    CONST robtarget point_414_contact:=[[206,145,134.5],[0,0,1,0],[0, 0, 0, 0],[9E+09,9E+09,9E+09,9E+09,9E+09,9E+09]];
    CONST robtarget point_415_contact:=[[206,137,134.5],[0,0,1,0],[0, 0, 0, 0],[9E+09,9E+09,9E+09,9E+09,9E+09,9E+09]];
    CONST robtarget point_415_clearance:=[[206,137,149.5],[0,0,1,0],[0, 0, 0, 0],[9E+09,9E+09,9E+09,9E+09,9E+09,9E+09]];
    CONST robtarget point_416_clearance:=[[237,138,149.5],[0,0,1,0],[0, 0, 0, 0],[9E+09,9E+09,9E+09,9E+09,9E+09,9E+09]];
    CONST robtarget point_416_contact:=[[237,138,134.5],[0,0,1,0],[0, 0, 0, 0],[9E+09,9E+09,9E+09,9E+09,9E+09,9E+09]];
    CONST robtarget point_417_contact:=[[240,137,134.5],[0,0,1,0],[0, 0, 0, 0],[9E+09,9E+09,9E+09,9E+09,9E+09,9E+09]];
    CONST robtarget point_417_clearance:=[[240,137,149.5],[0,0,1,0],[0, 0, 0, 0],[9E+09,9E+09,9E+09,9E+09,9E+09,9E+09]];
    CONST robtarget point_418_clearance:=[[348,137,149.5],[0,0,1,0],[0, 0, 0, 0],[9E+09,9E+09,9E+09,9E+09,9E+09,9E+09]];
    CONST robtarget point_418_contact:=[[348,137,134.5],[0,0,1,0],[0, 0, 0, 0],[9E+09,9E+09,9E+09,9E+09,9E+09,9E+09]];
    CONST robtarget point_419_contact:=[[363,145,134.5],[0,0,1,0],[0, 0, 0, 0],[9E+09,9E+09,9E+09,9E+09,9E+09,9E+09]];
    CONST robtarget point_419_clearance:=[[363,145,149.5],[0,0,1,0],[0, 0, 0, 0],[9E+09,9E+09,9E+09,9E+09,9E+09,9E+09]];
    CONST robtarget point_420_clearance:=[[399,156,149.5],[0,0,1,0],[0, 0, 0, 0],[9E+09,9E+09,9E+09,9E+09,9E+09,9E+09]];
    CONST robtarget point_420_contact:=[[399,156,134.5],[0,0,1,0],[0, 0, 0, 0],[9E+09,9E+09,9E+09,9E+09,9E+09,9E+09]];
    CONST robtarget point_421_contact:=[[402,137,134.5],[0,0,1,0],[0, 0, 0, 0],[9E+09,9E+09,9E+09,9E+09,9E+09,9E+09]];
    CONST robtarget point_421_clearance:=[[402,137,149.5],[0,0,1,0],[0, 0, 0, 0],[9E+09,9E+09,9E+09,9E+09,9E+09,9E+09]];
    CONST robtarget point_422_clearance:=[[144,140,149.5],[0,0,1,0],[0, 0, 0, 0],[9E+09,9E+09,9E+09,9E+09,9E+09,9E+09]];
    CONST robtarget point_422_contact:=[[144,140,134.5],[0,0,1,0],[0, 0, 0, 0],[9E+09,9E+09,9E+09,9E+09,9E+09,9E+09]];
    CONST robtarget point_423_contact:=[[159,145,134.5],[0,0,1,0],[0, 0, 0, 0],[9E+09,9E+09,9E+09,9E+09,9E+09,9E+09]];
    CONST robtarget point_423_clearance:=[[159,145,149.5],[0,0,1,0],[0, 0, 0, 0],[9E+09,9E+09,9E+09,9E+09,9E+09,9E+09]];
    CONST robtarget point_424_clearance:=[[249,145,149.5],[0,0,1,0],[0, 0, 0, 0],[9E+09,9E+09,9E+09,9E+09,9E+09,9E+09]];
    CONST robtarget point_424_contact:=[[249,145,134.5],[0,0,1,0],[0, 0, 0, 0],[9E+09,9E+09,9E+09,9E+09,9E+09,9E+09]];
    CONST robtarget point_425_contact:=[[256,139,134.5],[0,0,1,0],[0, 0, 0, 0],[9E+09,9E+09,9E+09,9E+09,9E+09,9E+09]];
    CONST robtarget point_425_clearance:=[[256,139,149.5],[0,0,1,0],[0, 0, 0, 0],[9E+09,9E+09,9E+09,9E+09,9E+09,9E+09]];
    CONST robtarget point_426_clearance:=[[316,140,149.5],[0,0,1,0],[0, 0, 0, 0],[9E+09,9E+09,9E+09,9E+09,9E+09,9E+09]];
    CONST robtarget point_426_contact:=[[316,140,134.5],[0,0,1,0],[0, 0, 0, 0],[9E+09,9E+09,9E+09,9E+09,9E+09,9E+09]];
    CONST robtarget point_427_contact:=[[312,141,134.5],[0,0,1,0],[0, 0, 0, 0],[9E+09,9E+09,9E+09,9E+09,9E+09,9E+09]];
    CONST robtarget point_427_clearance:=[[312,141,149.5],[0,0,1,0],[0, 0, 0, 0],[9E+09,9E+09,9E+09,9E+09,9E+09,9E+09]];
    CONST robtarget point_428_clearance:=[[313,144,149.5],[0,0,1,0],[0, 0, 0, 0],[9E+09,9E+09,9E+09,9E+09,9E+09,9E+09]];
    CONST robtarget point_428_contact:=[[313,144,134.5],[0,0,1,0],[0, 0, 0, 0],[9E+09,9E+09,9E+09,9E+09,9E+09,9E+09]];
    CONST robtarget point_429_contact:=[[322,138,134.5],[0,0,1,0],[0, 0, 0, 0],[9E+09,9E+09,9E+09,9E+09,9E+09,9E+09]];
    CONST robtarget point_429_clearance:=[[322,138,149.5],[0,0,1,0],[0, 0, 0, 0],[9E+09,9E+09,9E+09,9E+09,9E+09,9E+09]];
    CONST robtarget point_430_clearance:=[[368,140,149.5],[0,0,1,0],[0, 0, 0, 0],[9E+09,9E+09,9E+09,9E+09,9E+09,9E+09]];
    CONST robtarget point_430_contact:=[[368,140,134.5],[0,0,1,0],[0, 0, 0, 0],[9E+09,9E+09,9E+09,9E+09,9E+09,9E+09]];
    CONST robtarget point_431_contact:=[[371,139,134.5],[0,0,1,0],[0, 0, 0, 0],[9E+09,9E+09,9E+09,9E+09,9E+09,9E+09]];
    CONST robtarget point_431_clearance:=[[371,139,149.5],[0,0,1,0],[0, 0, 0, 0],[9E+09,9E+09,9E+09,9E+09,9E+09,9E+09]];
    CONST robtarget point_432_clearance:=[[306,146,149.5],[0,0,1,0],[0, 0, 0, 0],[9E+09,9E+09,9E+09,9E+09,9E+09,9E+09]];
    CONST robtarget point_432_contact:=[[306,146,134.5],[0,0,1,0],[0, 0, 0, 0],[9E+09,9E+09,9E+09,9E+09,9E+09,9E+09]];
    CONST robtarget point_433_contact:=[[299,140,134.5],[0,0,1,0],[0, 0, 0, 0],[9E+09,9E+09,9E+09,9E+09,9E+09,9E+09]];
    CONST robtarget point_433_clearance:=[[299,140,149.5],[0,0,1,0],[0, 0, 0, 0],[9E+09,9E+09,9E+09,9E+09,9E+09,9E+09]];
    CONST robtarget point_434_clearance:=[[411,141,149.5],[0,0,1,0],[0, 0, 0, 0],[9E+09,9E+09,9E+09,9E+09,9E+09,9E+09]];
    CONST robtarget point_434_contact:=[[411,141,134.5],[0,0,1,0],[0, 0, 0, 0],[9E+09,9E+09,9E+09,9E+09,9E+09,9E+09]];
    CONST robtarget point_435_contact:=[[409,155,134.5],[0,0,1,0],[0, 0, 0, 0],[9E+09,9E+09,9E+09,9E+09,9E+09,9E+09]];
    CONST robtarget point_435_clearance:=[[409,155,149.5],[0,0,1,0],[0, 0, 0, 0],[9E+09,9E+09,9E+09,9E+09,9E+09,9E+09]];
    CONST robtarget point_436_clearance:=[[160,143,149.5],[0,0,1,0],[0, 0, 0, 0],[9E+09,9E+09,9E+09,9E+09,9E+09,9E+09]];
    CONST robtarget point_436_contact:=[[160,143,134.5],[0,0,1,0],[0, 0, 0, 0],[9E+09,9E+09,9E+09,9E+09,9E+09,9E+09]];
    CONST robtarget point_437_contact:=[[160,162,134.5],[0,0,1,0],[0, 0, 0, 0],[9E+09,9E+09,9E+09,9E+09,9E+09,9E+09]];
    CONST robtarget point_437_clearance:=[[160,162,149.5],[0,0,1,0],[0, 0, 0, 0],[9E+09,9E+09,9E+09,9E+09,9E+09,9E+09]];
    CONST robtarget point_438_clearance:=[[316,147,149.5],[0,0,1,0],[0, 0, 0, 0],[9E+09,9E+09,9E+09,9E+09,9E+09,9E+09]];
    CONST robtarget point_438_contact:=[[316,147,134.5],[0,0,1,0],[0, 0, 0, 0],[9E+09,9E+09,9E+09,9E+09,9E+09,9E+09]];
    CONST robtarget point_439_contact:=[[306,146,134.5],[0,0,1,0],[0, 0, 0, 0],[9E+09,9E+09,9E+09,9E+09,9E+09,9E+09]];
    CONST robtarget point_439_clearance:=[[306,146,149.5],[0,0,1,0],[0, 0, 0, 0],[9E+09,9E+09,9E+09,9E+09,9E+09,9E+09]];
    CONST robtarget point_440_clearance:=[[435,170,149.5],[0,0,1,0],[0, 0, 0, 0],[9E+09,9E+09,9E+09,9E+09,9E+09,9E+09]];
    CONST robtarget point_440_contact:=[[435,170,134.5],[0,0,1,0],[0, 0, 0, 0],[9E+09,9E+09,9E+09,9E+09,9E+09,9E+09]];
    CONST robtarget point_441_contact:=[[433,143,134.5],[0,0,1,0],[0, 0, 0, 0],[9E+09,9E+09,9E+09,9E+09,9E+09,9E+09]];
    CONST robtarget point_441_clearance:=[[433,143,149.5],[0,0,1,0],[0, 0, 0, 0],[9E+09,9E+09,9E+09,9E+09,9E+09,9E+09]];
    CONST robtarget point_442_clearance:=[[326,146,149.5],[0,0,1,0],[0, 0, 0, 0],[9E+09,9E+09,9E+09,9E+09,9E+09,9E+09]];
    CONST robtarget point_442_contact:=[[326,146,134.5],[0,0,1,0],[0, 0, 0, 0],[9E+09,9E+09,9E+09,9E+09,9E+09,9E+09]];
    CONST robtarget point_443_contact:=[[317,146,134.5],[0,0,1,0],[0, 0, 0, 0],[9E+09,9E+09,9E+09,9E+09,9E+09,9E+09]];
    CONST robtarget point_443_clearance:=[[317,146,149.5],[0,0,1,0],[0, 0, 0, 0],[9E+09,9E+09,9E+09,9E+09,9E+09,9E+09]];
    CONST robtarget point_444_clearance:=[[378,183,149.5],[0,0,1,0],[0, 0, 0, 0],[9E+09,9E+09,9E+09,9E+09,9E+09,9E+09]];
    CONST robtarget point_444_contact:=[[378,183,134.5],[0,0,1,0],[0, 0, 0, 0],[9E+09,9E+09,9E+09,9E+09,9E+09,9E+09]];
    CONST robtarget point_445_contact:=[[391,144,134.5],[0,0,1,0],[0, 0, 0, 0],[9E+09,9E+09,9E+09,9E+09,9E+09,9E+09]];
    CONST robtarget point_445_clearance:=[[391,144,149.5],[0,0,1,0],[0, 0, 0, 0],[9E+09,9E+09,9E+09,9E+09,9E+09,9E+09]];
    CONST robtarget point_446_clearance:=[[166,147,149.5],[0,0,1,0],[0, 0, 0, 0],[9E+09,9E+09,9E+09,9E+09,9E+09,9E+09]];
    CONST robtarget point_446_contact:=[[166,147,134.5],[0,0,1,0],[0, 0, 0, 0],[9E+09,9E+09,9E+09,9E+09,9E+09,9E+09]];
    CONST robtarget point_447_contact:=[[176,150,134.5],[0,0,1,0],[0, 0, 0, 0],[9E+09,9E+09,9E+09,9E+09,9E+09,9E+09]];
    CONST robtarget point_447_clearance:=[[176,150,149.5],[0,0,1,0],[0, 0, 0, 0],[9E+09,9E+09,9E+09,9E+09,9E+09,9E+09]];
    CONST robtarget point_448_clearance:=[[198,172,149.5],[0,0,1,0],[0, 0, 0, 0],[9E+09,9E+09,9E+09,9E+09,9E+09,9E+09]];
    CONST robtarget point_448_contact:=[[198,172,134.5],[0,0,1,0],[0, 0, 0, 0],[9E+09,9E+09,9E+09,9E+09,9E+09,9E+09]];
    CONST robtarget point_449_contact:=[[198,146,134.5],[0,0,1,0],[0, 0, 0, 0],[9E+09,9E+09,9E+09,9E+09,9E+09,9E+09]];
    CONST robtarget point_449_clearance:=[[198,146,149.5],[0,0,1,0],[0, 0, 0, 0],[9E+09,9E+09,9E+09,9E+09,9E+09,9E+09]];
    CONST robtarget point_450_clearance:=[[213,226,149.5],[0,0,1,0],[0, 0, 0, 0],[9E+09,9E+09,9E+09,9E+09,9E+09,9E+09]];
    CONST robtarget point_450_contact:=[[213,226,134.5],[0,0,1,0],[0, 0, 0, 0],[9E+09,9E+09,9E+09,9E+09,9E+09,9E+09]];
    CONST robtarget point_451_contact:=[[206,146,134.5],[0,0,1,0],[0, 0, 0, 0],[9E+09,9E+09,9E+09,9E+09,9E+09,9E+09]];
    CONST robtarget point_451_clearance:=[[206,146,149.5],[0,0,1,0],[0, 0, 0, 0],[9E+09,9E+09,9E+09,9E+09,9E+09,9E+09]];
    CONST robtarget point_452_clearance:=[[165,163,149.5],[0,0,1,0],[0, 0, 0, 0],[9E+09,9E+09,9E+09,9E+09,9E+09,9E+09]];
    CONST robtarget point_452_contact:=[[165,163,134.5],[0,0,1,0],[0, 0, 0, 0],[9E+09,9E+09,9E+09,9E+09,9E+09,9E+09]];
    CONST robtarget point_453_contact:=[[165,150,134.5],[0,0,1,0],[0, 0, 0, 0],[9E+09,9E+09,9E+09,9E+09,9E+09,9E+09]];
    CONST robtarget point_453_clearance:=[[165,150,149.5],[0,0,1,0],[0, 0, 0, 0],[9E+09,9E+09,9E+09,9E+09,9E+09,9E+09]];
    CONST robtarget point_454_clearance:=[[188,150,149.5],[0,0,1,0],[0, 0, 0, 0],[9E+09,9E+09,9E+09,9E+09,9E+09,9E+09]];
    CONST robtarget point_454_contact:=[[188,150,134.5],[0,0,1,0],[0, 0, 0, 0],[9E+09,9E+09,9E+09,9E+09,9E+09,9E+09]];
    CONST robtarget point_455_contact:=[[188,170,134.5],[0,0,1,0],[0, 0, 0, 0],[9E+09,9E+09,9E+09,9E+09,9E+09,9E+09]];
    CONST robtarget point_455_clearance:=[[188,170,149.5],[0,0,1,0],[0, 0, 0, 0],[9E+09,9E+09,9E+09,9E+09,9E+09,9E+09]];
    CONST robtarget point_456_clearance:=[[230,150,149.5],[0,0,1,0],[0, 0, 0, 0],[9E+09,9E+09,9E+09,9E+09,9E+09,9E+09]];
    CONST robtarget point_456_contact:=[[230,150,134.5],[0,0,1,0],[0, 0, 0, 0],[9E+09,9E+09,9E+09,9E+09,9E+09,9E+09]];
    CONST robtarget point_457_contact:=[[237,168,134.5],[0,0,1,0],[0, 0, 0, 0],[9E+09,9E+09,9E+09,9E+09,9E+09,9E+09]];
    CONST robtarget point_457_clearance:=[[237,168,149.5],[0,0,1,0],[0, 0, 0, 0],[9E+09,9E+09,9E+09,9E+09,9E+09,9E+09]];
    CONST robtarget point_458_clearance:=[[266,154,149.5],[0,0,1,0],[0, 0, 0, 0],[9E+09,9E+09,9E+09,9E+09,9E+09,9E+09]];
    CONST robtarget point_458_contact:=[[266,154,134.5],[0,0,1,0],[0, 0, 0, 0],[9E+09,9E+09,9E+09,9E+09,9E+09,9E+09]];
    CONST robtarget point_459_contact:=[[343,158,134.5],[0,0,1,0],[0, 0, 0, 0],[9E+09,9E+09,9E+09,9E+09,9E+09,9E+09]];
    CONST robtarget point_459_clearance:=[[343,158,149.5],[0,0,1,0],[0, 0, 0, 0],[9E+09,9E+09,9E+09,9E+09,9E+09,9E+09]];
    CONST robtarget point_460_clearance:=[[357,162,149.5],[0,0,1,0],[0, 0, 0, 0],[9E+09,9E+09,9E+09,9E+09,9E+09,9E+09]];
    CONST robtarget point_460_contact:=[[357,162,134.5],[0,0,1,0],[0, 0, 0, 0],[9E+09,9E+09,9E+09,9E+09,9E+09,9E+09]];
    CONST robtarget point_461_contact:=[[344,149,134.5],[0,0,1,0],[0, 0, 0, 0],[9E+09,9E+09,9E+09,9E+09,9E+09,9E+09]];
    CONST robtarget point_461_clearance:=[[344,149,149.5],[0,0,1,0],[0, 0, 0, 0],[9E+09,9E+09,9E+09,9E+09,9E+09,9E+09]];
    CONST robtarget point_462_clearance:=[[179,151,149.5],[0,0,1,0],[0, 0, 0, 0],[9E+09,9E+09,9E+09,9E+09,9E+09,9E+09]];
    CONST robtarget point_462_contact:=[[179,151,134.5],[0,0,1,0],[0, 0, 0, 0],[9E+09,9E+09,9E+09,9E+09,9E+09,9E+09]];
    CONST robtarget point_463_contact:=[[179,167,134.5],[0,0,1,0],[0, 0, 0, 0],[9E+09,9E+09,9E+09,9E+09,9E+09,9E+09]];
    CONST robtarget point_463_clearance:=[[179,167,149.5],[0,0,1,0],[0, 0, 0, 0],[9E+09,9E+09,9E+09,9E+09,9E+09,9E+09]];
    CONST robtarget point_464_clearance:=[[413,187,149.5],[0,0,1,0],[0, 0, 0, 0],[9E+09,9E+09,9E+09,9E+09,9E+09,9E+09]];
    CONST robtarget point_464_contact:=[[413,187,134.5],[0,0,1,0],[0, 0, 0, 0],[9E+09,9E+09,9E+09,9E+09,9E+09,9E+09]];
    CONST robtarget point_465_contact:=[[415,151,134.5],[0,0,1,0],[0, 0, 0, 0],[9E+09,9E+09,9E+09,9E+09,9E+09,9E+09]];
    CONST robtarget point_465_clearance:=[[415,151,149.5],[0,0,1,0],[0, 0, 0, 0],[9E+09,9E+09,9E+09,9E+09,9E+09,9E+09]];
    CONST robtarget point_466_clearance:=[[257,154,149.5],[0,0,1,0],[0, 0, 0, 0],[9E+09,9E+09,9E+09,9E+09,9E+09,9E+09]];
    CONST robtarget point_466_contact:=[[257,154,134.5],[0,0,1,0],[0, 0, 0, 0],[9E+09,9E+09,9E+09,9E+09,9E+09,9E+09]];
    CONST robtarget point_467_contact:=[[241,160,134.5],[0,0,1,0],[0, 0, 0, 0],[9E+09,9E+09,9E+09,9E+09,9E+09,9E+09]];
    CONST robtarget point_467_clearance:=[[241,160,149.5],[0,0,1,0],[0, 0, 0, 0],[9E+09,9E+09,9E+09,9E+09,9E+09,9E+09]];
    CONST robtarget point_468_clearance:=[[260,158,149.5],[0,0,1,0],[0, 0, 0, 0],[9E+09,9E+09,9E+09,9E+09,9E+09,9E+09]];
    CONST robtarget point_468_contact:=[[260,158,134.5],[0,0,1,0],[0, 0, 0, 0],[9E+09,9E+09,9E+09,9E+09,9E+09,9E+09]];
    CONST robtarget point_469_contact:=[[265,153,134.5],[0,0,1,0],[0, 0, 0, 0],[9E+09,9E+09,9E+09,9E+09,9E+09,9E+09]];
    CONST robtarget point_469_clearance:=[[265,153,149.5],[0,0,1,0],[0, 0, 0, 0],[9E+09,9E+09,9E+09,9E+09,9E+09,9E+09]];
    CONST robtarget point_470_clearance:=[[410,154,149.5],[0,0,1,0],[0, 0, 0, 0],[9E+09,9E+09,9E+09,9E+09,9E+09,9E+09]];
    CONST robtarget point_470_contact:=[[410,154,134.5],[0,0,1,0],[0, 0, 0, 0],[9E+09,9E+09,9E+09,9E+09,9E+09,9E+09]];
    CONST robtarget point_471_contact:=[[398,192,134.5],[0,0,1,0],[0, 0, 0, 0],[9E+09,9E+09,9E+09,9E+09,9E+09,9E+09]];
    CONST robtarget point_471_clearance:=[[398,192,149.5],[0,0,1,0],[0, 0, 0, 0],[9E+09,9E+09,9E+09,9E+09,9E+09,9E+09]];
    CONST robtarget point_472_clearance:=[[161,164,149.5],[0,0,1,0],[0, 0, 0, 0],[9E+09,9E+09,9E+09,9E+09,9E+09,9E+09]];
    CONST robtarget point_472_contact:=[[161,164,134.5],[0,0,1,0],[0, 0, 0, 0],[9E+09,9E+09,9E+09,9E+09,9E+09,9E+09]];
    CONST robtarget point_473_contact:=[[145,159,134.5],[0,0,1,0],[0, 0, 0, 0],[9E+09,9E+09,9E+09,9E+09,9E+09,9E+09]];
    CONST robtarget point_473_clearance:=[[145,159,149.5],[0,0,1,0],[0, 0, 0, 0],[9E+09,9E+09,9E+09,9E+09,9E+09,9E+09]];
    CONST robtarget point_474_clearance:=[[191,182,149.5],[0,0,1,0],[0, 0, 0, 0],[9E+09,9E+09,9E+09,9E+09,9E+09,9E+09]];
    CONST robtarget point_474_contact:=[[191,182,134.5],[0,0,1,0],[0, 0, 0, 0],[9E+09,9E+09,9E+09,9E+09,9E+09,9E+09]];
    CONST robtarget point_475_contact:=[[192,157,134.5],[0,0,1,0],[0, 0, 0, 0],[9E+09,9E+09,9E+09,9E+09,9E+09,9E+09]];
    CONST robtarget point_475_clearance:=[[192,157,149.5],[0,0,1,0],[0, 0, 0, 0],[9E+09,9E+09,9E+09,9E+09,9E+09,9E+09]];
    CONST robtarget point_476_clearance:=[[218,178,149.5],[0,0,1,0],[0, 0, 0, 0],[9E+09,9E+09,9E+09,9E+09,9E+09,9E+09]];
    CONST robtarget point_476_contact:=[[218,178,134.5],[0,0,1,0],[0, 0, 0, 0],[9E+09,9E+09,9E+09,9E+09,9E+09,9E+09]];
    CONST robtarget point_477_contact:=[[219,157,134.5],[0,0,1,0],[0, 0, 0, 0],[9E+09,9E+09,9E+09,9E+09,9E+09,9E+09]];
    CONST robtarget point_477_clearance:=[[219,157,149.5],[0,0,1,0],[0, 0, 0, 0],[9E+09,9E+09,9E+09,9E+09,9E+09,9E+09]];
    CONST robtarget point_478_clearance:=[[315,163,149.5],[0,0,1,0],[0, 0, 0, 0],[9E+09,9E+09,9E+09,9E+09,9E+09,9E+09]];
    CONST robtarget point_478_contact:=[[315,163,134.5],[0,0,1,0],[0, 0, 0, 0],[9E+09,9E+09,9E+09,9E+09,9E+09,9E+09]];
    CONST robtarget point_479_contact:=[[257,160,134.5],[0,0,1,0],[0, 0, 0, 0],[9E+09,9E+09,9E+09,9E+09,9E+09,9E+09]];
    CONST robtarget point_479_clearance:=[[257,160,149.5],[0,0,1,0],[0, 0, 0, 0],[9E+09,9E+09,9E+09,9E+09,9E+09,9E+09]];
    CONST robtarget point_480_clearance:=[[395,187,149.5],[0,0,1,0],[0, 0, 0, 0],[9E+09,9E+09,9E+09,9E+09,9E+09,9E+09]];
    CONST robtarget point_480_contact:=[[395,187,134.5],[0,0,1,0],[0, 0, 0, 0],[9E+09,9E+09,9E+09,9E+09,9E+09,9E+09]];
    CONST robtarget point_481_contact:=[[401,160,134.5],[0,0,1,0],[0, 0, 0, 0],[9E+09,9E+09,9E+09,9E+09,9E+09,9E+09]];
    CONST robtarget point_481_clearance:=[[401,160,149.5],[0,0,1,0],[0, 0, 0, 0],[9E+09,9E+09,9E+09,9E+09,9E+09,9E+09]];
    CONST robtarget point_482_clearance:=[[285,172,149.5],[0,0,1,0],[0, 0, 0, 0],[9E+09,9E+09,9E+09,9E+09,9E+09,9E+09]];
    CONST robtarget point_482_contact:=[[285,172,134.5],[0,0,1,0],[0, 0, 0, 0],[9E+09,9E+09,9E+09,9E+09,9E+09,9E+09]];
    CONST robtarget point_483_contact:=[[271,161,134.5],[0,0,1,0],[0, 0, 0, 0],[9E+09,9E+09,9E+09,9E+09,9E+09,9E+09]];
    CONST robtarget point_483_clearance:=[[271,161,149.5],[0,0,1,0],[0, 0, 0, 0],[9E+09,9E+09,9E+09,9E+09,9E+09,9E+09]];
    CONST robtarget point_484_clearance:=[[356,164,149.5],[0,0,1,0],[0, 0, 0, 0],[9E+09,9E+09,9E+09,9E+09,9E+09,9E+09]];
    CONST robtarget point_484_contact:=[[356,164,134.5],[0,0,1,0],[0, 0, 0, 0],[9E+09,9E+09,9E+09,9E+09,9E+09,9E+09]];
    CONST robtarget point_485_contact:=[[363,162,134.5],[0,0,1,0],[0, 0, 0, 0],[9E+09,9E+09,9E+09,9E+09,9E+09,9E+09]];
    CONST robtarget point_485_clearance:=[[363,162,149.5],[0,0,1,0],[0, 0, 0, 0],[9E+09,9E+09,9E+09,9E+09,9E+09,9E+09]];
    CONST robtarget point_486_clearance:=[[347,164,149.5],[0,0,1,0],[0, 0, 0, 0],[9E+09,9E+09,9E+09,9E+09,9E+09,9E+09]];
    CONST robtarget point_486_contact:=[[347,164,134.5],[0,0,1,0],[0, 0, 0, 0],[9E+09,9E+09,9E+09,9E+09,9E+09,9E+09]];
    CONST robtarget point_487_contact:=[[316,163,134.5],[0,0,1,0],[0, 0, 0, 0],[9E+09,9E+09,9E+09,9E+09,9E+09,9E+09]];
    CONST robtarget point_487_clearance:=[[316,163,149.5],[0,0,1,0],[0, 0, 0, 0],[9E+09,9E+09,9E+09,9E+09,9E+09,9E+09]];
    CONST robtarget point_488_clearance:=[[176,169,149.5],[0,0,1,0],[0, 0, 0, 0],[9E+09,9E+09,9E+09,9E+09,9E+09,9E+09]];
    CONST robtarget point_488_contact:=[[176,169,134.5],[0,0,1,0],[0, 0, 0, 0],[9E+09,9E+09,9E+09,9E+09,9E+09,9E+09]];
    CONST robtarget point_489_contact:=[[171,164,134.5],[0,0,1,0],[0, 0, 0, 0],[9E+09,9E+09,9E+09,9E+09,9E+09,9E+09]];
    CONST robtarget point_489_clearance:=[[171,164,149.5],[0,0,1,0],[0, 0, 0, 0],[9E+09,9E+09,9E+09,9E+09,9E+09,9E+09]];
    CONST robtarget point_490_clearance:=[[203,164,149.5],[0,0,1,0],[0, 0, 0, 0],[9E+09,9E+09,9E+09,9E+09,9E+09,9E+09]];
    CONST robtarget point_490_contact:=[[203,164,134.5],[0,0,1,0],[0, 0, 0, 0],[9E+09,9E+09,9E+09,9E+09,9E+09,9E+09]];
    CONST robtarget point_491_contact:=[[206,185,134.5],[0,0,1,0],[0, 0, 0, 0],[9E+09,9E+09,9E+09,9E+09,9E+09,9E+09]];
    CONST robtarget point_491_clearance:=[[206,185,149.5],[0,0,1,0],[0, 0, 0, 0],[9E+09,9E+09,9E+09,9E+09,9E+09,9E+09]];
    CONST robtarget point_492_clearance:=[[331,167,149.5],[0,0,1,0],[0, 0, 0, 0],[9E+09,9E+09,9E+09,9E+09,9E+09,9E+09]];
    CONST robtarget point_492_contact:=[[331,167,134.5],[0,0,1,0],[0, 0, 0, 0],[9E+09,9E+09,9E+09,9E+09,9E+09,9E+09]];
    CONST robtarget point_493_contact:=[[340,168,134.5],[0,0,1,0],[0, 0, 0, 0],[9E+09,9E+09,9E+09,9E+09,9E+09,9E+09]];
    CONST robtarget point_493_clearance:=[[340,168,149.5],[0,0,1,0],[0, 0, 0, 0],[9E+09,9E+09,9E+09,9E+09,9E+09,9E+09]];
    CONST robtarget point_494_clearance:=[[396,165,149.5],[0,0,1,0],[0, 0, 0, 0],[9E+09,9E+09,9E+09,9E+09,9E+09,9E+09]];
    CONST robtarget point_494_contact:=[[396,165,134.5],[0,0,1,0],[0, 0, 0, 0],[9E+09,9E+09,9E+09,9E+09,9E+09,9E+09]];
    CONST robtarget point_495_contact:=[[393,183,134.5],[0,0,1,0],[0, 0, 0, 0],[9E+09,9E+09,9E+09,9E+09,9E+09,9E+09]];
    CONST robtarget point_495_clearance:=[[393,183,149.5],[0,0,1,0],[0, 0, 0, 0],[9E+09,9E+09,9E+09,9E+09,9E+09,9E+09]];
    CONST robtarget point_496_clearance:=[[286,166,149.5],[0,0,1,0],[0, 0, 0, 0],[9E+09,9E+09,9E+09,9E+09,9E+09,9E+09]];
    CONST robtarget point_496_contact:=[[286,166,134.5],[0,0,1,0],[0, 0, 0, 0],[9E+09,9E+09,9E+09,9E+09,9E+09,9E+09]];
    CONST robtarget point_497_contact:=[[306,170,134.5],[0,0,1,0],[0, 0, 0, 0],[9E+09,9E+09,9E+09,9E+09,9E+09,9E+09]];
    CONST robtarget point_497_clearance:=[[306,170,149.5],[0,0,1,0],[0, 0, 0, 0],[9E+09,9E+09,9E+09,9E+09,9E+09,9E+09]];
    CONST robtarget point_498_clearance:=[[364,171,149.5],[0,0,1,0],[0, 0, 0, 0],[9E+09,9E+09,9E+09,9E+09,9E+09,9E+09]];
    CONST robtarget point_498_contact:=[[364,171,134.5],[0,0,1,0],[0, 0, 0, 0],[9E+09,9E+09,9E+09,9E+09,9E+09,9E+09]];
    CONST robtarget point_499_contact:=[[367,166,134.5],[0,0,1,0],[0, 0, 0, 0],[9E+09,9E+09,9E+09,9E+09,9E+09,9E+09]];
    CONST robtarget point_499_clearance:=[[367,166,149.5],[0,0,1,0],[0, 0, 0, 0],[9E+09,9E+09,9E+09,9E+09,9E+09,9E+09]];
    CONST robtarget point_500_clearance:=[[425,166,149.5],[0,0,1,0],[0, 0, 0, 0],[9E+09,9E+09,9E+09,9E+09,9E+09,9E+09]];
    CONST robtarget point_500_contact:=[[425,166,134.5],[0,0,1,0],[0, 0, 0, 0],[9E+09,9E+09,9E+09,9E+09,9E+09,9E+09]];
    CONST robtarget point_501_contact:=[[421,199,134.5],[0,0,1,0],[0, 0, 0, 0],[9E+09,9E+09,9E+09,9E+09,9E+09,9E+09]];
    CONST robtarget point_501_clearance:=[[421,199,149.5],[0,0,1,0],[0, 0, 0, 0],[9E+09,9E+09,9E+09,9E+09,9E+09,9E+09]];
    CONST robtarget point_502_clearance:=[[425,196,149.5],[0,0,1,0],[0, 0, 0, 0],[9E+09,9E+09,9E+09,9E+09,9E+09,9E+09]];
    CONST robtarget point_502_contact:=[[425,196,134.5],[0,0,1,0],[0, 0, 0, 0],[9E+09,9E+09,9E+09,9E+09,9E+09,9E+09]];
    CONST robtarget point_503_contact:=[[428,166,134.5],[0,0,1,0],[0, 0, 0, 0],[9E+09,9E+09,9E+09,9E+09,9E+09,9E+09]];
    CONST robtarget point_503_clearance:=[[428,166,149.5],[0,0,1,0],[0, 0, 0, 0],[9E+09,9E+09,9E+09,9E+09,9E+09,9E+09]];
    CONST robtarget point_504_clearance:=[[307,169,149.5],[0,0,1,0],[0, 0, 0, 0],[9E+09,9E+09,9E+09,9E+09,9E+09,9E+09]];
    CONST robtarget point_504_contact:=[[307,169,134.5],[0,0,1,0],[0, 0, 0, 0],[9E+09,9E+09,9E+09,9E+09,9E+09,9E+09]];
    CONST robtarget point_505_contact:=[[323,168,134.5],[0,0,1,0],[0, 0, 0, 0],[9E+09,9E+09,9E+09,9E+09,9E+09,9E+09]];
    CONST robtarget point_505_clearance:=[[323,168,149.5],[0,0,1,0],[0, 0, 0, 0],[9E+09,9E+09,9E+09,9E+09,9E+09,9E+09]];
    CONST robtarget point_506_clearance:=[[330,168,149.5],[0,0,1,0],[0, 0, 0, 0],[9E+09,9E+09,9E+09,9E+09,9E+09,9E+09]];
    CONST robtarget point_506_contact:=[[330,168,134.5],[0,0,1,0],[0, 0, 0, 0],[9E+09,9E+09,9E+09,9E+09,9E+09,9E+09]];
    CONST robtarget point_507_contact:=[[319,174,134.5],[0,0,1,0],[0, 0, 0, 0],[9E+09,9E+09,9E+09,9E+09,9E+09,9E+09]];
    CONST robtarget point_507_clearance:=[[319,174,149.5],[0,0,1,0],[0, 0, 0, 0],[9E+09,9E+09,9E+09,9E+09,9E+09,9E+09]];
    CONST robtarget point_508_clearance:=[[138,170,149.5],[0,0,1,0],[0, 0, 0, 0],[9E+09,9E+09,9E+09,9E+09,9E+09,9E+09]];
    CONST robtarget point_508_contact:=[[138,170,134.5],[0,0,1,0],[0, 0, 0, 0],[9E+09,9E+09,9E+09,9E+09,9E+09,9E+09]];
    CONST robtarget point_509_contact:=[[159,174,134.5],[0,0,1,0],[0, 0, 0, 0],[9E+09,9E+09,9E+09,9E+09,9E+09,9E+09]];
    CONST robtarget point_509_clearance:=[[159,174,149.5],[0,0,1,0],[0, 0, 0, 0],[9E+09,9E+09,9E+09,9E+09,9E+09,9E+09]];
    CONST robtarget point_510_clearance:=[[237,168,149.5],[0,0,1,0],[0, 0, 0, 0],[9E+09,9E+09,9E+09,9E+09,9E+09,9E+09]];
    CONST robtarget point_510_contact:=[[237,168,134.5],[0,0,1,0],[0, 0, 0, 0],[9E+09,9E+09,9E+09,9E+09,9E+09,9E+09]];
    CONST robtarget point_511_contact:=[[238,176,134.5],[0,0,1,0],[0, 0, 0, 0],[9E+09,9E+09,9E+09,9E+09,9E+09,9E+09]];
    CONST robtarget point_511_clearance:=[[238,176,149.5],[0,0,1,0],[0, 0, 0, 0],[9E+09,9E+09,9E+09,9E+09,9E+09,9E+09]];
    CONST robtarget point_512_clearance:=[[357,169,149.5],[0,0,1,0],[0, 0, 0, 0],[9E+09,9E+09,9E+09,9E+09,9E+09,9E+09]];
    CONST robtarget point_512_contact:=[[357,169,134.5],[0,0,1,0],[0, 0, 0, 0],[9E+09,9E+09,9E+09,9E+09,9E+09,9E+09]];
    CONST robtarget point_513_contact:=[[360,172,134.5],[0,0,1,0],[0, 0, 0, 0],[9E+09,9E+09,9E+09,9E+09,9E+09,9E+09]];
    CONST robtarget point_513_clearance:=[[360,172,149.5],[0,0,1,0],[0, 0, 0, 0],[9E+09,9E+09,9E+09,9E+09,9E+09,9E+09]];
    CONST robtarget point_514_clearance:=[[412,168,149.5],[0,0,1,0],[0, 0, 0, 0],[9E+09,9E+09,9E+09,9E+09,9E+09,9E+09]];
    CONST robtarget point_514_contact:=[[412,168,134.5],[0,0,1,0],[0, 0, 0, 0],[9E+09,9E+09,9E+09,9E+09,9E+09,9E+09]];
    CONST robtarget point_515_contact:=[[407,197,134.5],[0,0,1,0],[0, 0, 0, 0],[9E+09,9E+09,9E+09,9E+09,9E+09,9E+09]];
    CONST robtarget point_515_clearance:=[[407,197,149.5],[0,0,1,0],[0, 0, 0, 0],[9E+09,9E+09,9E+09,9E+09,9E+09,9E+09]];
    CONST robtarget point_516_clearance:=[[188,170,149.5],[0,0,1,0],[0, 0, 0, 0],[9E+09,9E+09,9E+09,9E+09,9E+09,9E+09]];
    CONST robtarget point_516_contact:=[[188,170,134.5],[0,0,1,0],[0, 0, 0, 0],[9E+09,9E+09,9E+09,9E+09,9E+09,9E+09]];
    CONST robtarget point_517_contact:=[[186,175,134.5],[0,0,1,0],[0, 0, 0, 0],[9E+09,9E+09,9E+09,9E+09,9E+09,9E+09]];
    CONST robtarget point_517_clearance:=[[186,175,149.5],[0,0,1,0],[0, 0, 0, 0],[9E+09,9E+09,9E+09,9E+09,9E+09,9E+09]];
    CONST robtarget point_518_clearance:=[[200,173,149.5],[0,0,1,0],[0, 0, 0, 0],[9E+09,9E+09,9E+09,9E+09,9E+09,9E+09]];
    CONST robtarget point_518_contact:=[[200,173,134.5],[0,0,1,0],[0, 0, 0, 0],[9E+09,9E+09,9E+09,9E+09,9E+09,9E+09]];
    CONST robtarget point_519_contact:=[[201,186,134.5],[0,0,1,0],[0, 0, 0, 0],[9E+09,9E+09,9E+09,9E+09,9E+09,9E+09]];
    CONST robtarget point_519_clearance:=[[201,186,149.5],[0,0,1,0],[0, 0, 0, 0],[9E+09,9E+09,9E+09,9E+09,9E+09,9E+09]];
    CONST robtarget point_520_clearance:=[[160,175,149.5],[0,0,1,0],[0, 0, 0, 0],[9E+09,9E+09,9E+09,9E+09,9E+09,9E+09]];
    CONST robtarget point_520_contact:=[[160,175,134.5],[0,0,1,0],[0, 0, 0, 0],[9E+09,9E+09,9E+09,9E+09,9E+09,9E+09]];
    CONST robtarget point_521_contact:=[[160,197,134.5],[0,0,1,0],[0, 0, 0, 0],[9E+09,9E+09,9E+09,9E+09,9E+09,9E+09]];
    CONST robtarget point_521_clearance:=[[160,197,149.5],[0,0,1,0],[0, 0, 0, 0],[9E+09,9E+09,9E+09,9E+09,9E+09,9E+09]];
    CONST robtarget point_522_clearance:=[[165,191,149.5],[0,0,1,0],[0, 0, 0, 0],[9E+09,9E+09,9E+09,9E+09,9E+09,9E+09]];
    CONST robtarget point_522_contact:=[[165,191,134.5],[0,0,1,0],[0, 0, 0, 0],[9E+09,9E+09,9E+09,9E+09,9E+09,9E+09]];
    CONST robtarget point_523_contact:=[[165,175,134.5],[0,0,1,0],[0, 0, 0, 0],[9E+09,9E+09,9E+09,9E+09,9E+09,9E+09]];
    CONST robtarget point_523_clearance:=[[165,175,149.5],[0,0,1,0],[0, 0, 0, 0],[9E+09,9E+09,9E+09,9E+09,9E+09,9E+09]];
    CONST robtarget point_524_clearance:=[[229,231,149.5],[0,0,1,0],[0, 0, 0, 0],[9E+09,9E+09,9E+09,9E+09,9E+09,9E+09]];
    CONST robtarget point_524_contact:=[[229,231,134.5],[0,0,1,0],[0, 0, 0, 0],[9E+09,9E+09,9E+09,9E+09,9E+09,9E+09]];
    CONST robtarget point_525_contact:=[[224,175,134.5],[0,0,1,0],[0, 0, 0, 0],[9E+09,9E+09,9E+09,9E+09,9E+09,9E+09]];
    CONST robtarget point_525_clearance:=[[224,175,149.5],[0,0,1,0],[0, 0, 0, 0],[9E+09,9E+09,9E+09,9E+09,9E+09,9E+09]];
    CONST robtarget point_526_clearance:=[[227,175,149.5],[0,0,1,0],[0, 0, 0, 0],[9E+09,9E+09,9E+09,9E+09,9E+09,9E+09]];
    CONST robtarget point_526_contact:=[[227,175,134.5],[0,0,1,0],[0, 0, 0, 0],[9E+09,9E+09,9E+09,9E+09,9E+09,9E+09]];
    CONST robtarget point_527_contact:=[[235,190,134.5],[0,0,1,0],[0, 0, 0, 0],[9E+09,9E+09,9E+09,9E+09,9E+09,9E+09]];
    CONST robtarget point_527_clearance:=[[235,190,149.5],[0,0,1,0],[0, 0, 0, 0],[9E+09,9E+09,9E+09,9E+09,9E+09,9E+09]];
    CONST robtarget point_528_clearance:=[[298,177,149.5],[0,0,1,0],[0, 0, 0, 0],[9E+09,9E+09,9E+09,9E+09,9E+09,9E+09]];
    CONST robtarget point_528_contact:=[[298,177,134.5],[0,0,1,0],[0, 0, 0, 0],[9E+09,9E+09,9E+09,9E+09,9E+09,9E+09]];
    CONST robtarget point_529_contact:=[[294,175,134.5],[0,0,1,0],[0, 0, 0, 0],[9E+09,9E+09,9E+09,9E+09,9E+09,9E+09]];
    CONST robtarget point_529_clearance:=[[294,175,149.5],[0,0,1,0],[0, 0, 0, 0],[9E+09,9E+09,9E+09,9E+09,9E+09,9E+09]];
    CONST robtarget point_530_clearance:=[[187,176,149.5],[0,0,1,0],[0, 0, 0, 0],[9E+09,9E+09,9E+09,9E+09,9E+09,9E+09]];
    CONST robtarget point_530_contact:=[[187,176,134.5],[0,0,1,0],[0, 0, 0, 0],[9E+09,9E+09,9E+09,9E+09,9E+09,9E+09]];
    CONST robtarget point_531_contact:=[[183,206,134.5],[0,0,1,0],[0, 0, 0, 0],[9E+09,9E+09,9E+09,9E+09,9E+09,9E+09]];
    CONST robtarget point_531_clearance:=[[183,206,149.5],[0,0,1,0],[0, 0, 0, 0],[9E+09,9E+09,9E+09,9E+09,9E+09,9E+09]];
    CONST robtarget point_532_clearance:=[[238,177,149.5],[0,0,1,0],[0, 0, 0, 0],[9E+09,9E+09,9E+09,9E+09,9E+09,9E+09]];
    CONST robtarget point_532_contact:=[[238,177,134.5],[0,0,1,0],[0, 0, 0, 0],[9E+09,9E+09,9E+09,9E+09,9E+09,9E+09]];
    CONST robtarget point_533_contact:=[[241,189,134.5],[0,0,1,0],[0, 0, 0, 0],[9E+09,9E+09,9E+09,9E+09,9E+09,9E+09]];
    CONST robtarget point_533_clearance:=[[241,189,149.5],[0,0,1,0],[0, 0, 0, 0],[9E+09,9E+09,9E+09,9E+09,9E+09,9E+09]];
    CONST robtarget point_534_clearance:=[[296,180,149.5],[0,0,1,0],[0, 0, 0, 0],[9E+09,9E+09,9E+09,9E+09,9E+09,9E+09]];
    CONST robtarget point_534_contact:=[[296,180,134.5],[0,0,1,0],[0, 0, 0, 0],[9E+09,9E+09,9E+09,9E+09,9E+09,9E+09]];
    CONST robtarget point_535_contact:=[[287,179,134.5],[0,0,1,0],[0, 0, 0, 0],[9E+09,9E+09,9E+09,9E+09,9E+09,9E+09]];
    CONST robtarget point_535_clearance:=[[287,179,149.5],[0,0,1,0],[0, 0, 0, 0],[9E+09,9E+09,9E+09,9E+09,9E+09,9E+09]];
    CONST robtarget point_536_clearance:=[[222,235,149.5],[0,0,1,0],[0, 0, 0, 0],[9E+09,9E+09,9E+09,9E+09,9E+09,9E+09]];
    CONST robtarget point_536_contact:=[[222,235,134.5],[0,0,1,0],[0, 0, 0, 0],[9E+09,9E+09,9E+09,9E+09,9E+09,9E+09]];
    CONST robtarget point_537_contact:=[[218,179,134.5],[0,0,1,0],[0, 0, 0, 0],[9E+09,9E+09,9E+09,9E+09,9E+09,9E+09]];
    CONST robtarget point_537_clearance:=[[218,179,149.5],[0,0,1,0],[0, 0, 0, 0],[9E+09,9E+09,9E+09,9E+09,9E+09,9E+09]];
    CONST robtarget point_538_clearance:=[[358,207,149.5],[0,0,1,0],[0, 0, 0, 0],[9E+09,9E+09,9E+09,9E+09,9E+09,9E+09]];
    CONST robtarget point_538_contact:=[[358,207,134.5],[0,0,1,0],[0, 0, 0, 0],[9E+09,9E+09,9E+09,9E+09,9E+09,9E+09]];
    CONST robtarget point_539_contact:=[[378,181,134.5],[0,0,1,0],[0, 0, 0, 0],[9E+09,9E+09,9E+09,9E+09,9E+09,9E+09]];
    CONST robtarget point_539_clearance:=[[378,181,149.5],[0,0,1,0],[0, 0, 0, 0],[9E+09,9E+09,9E+09,9E+09,9E+09,9E+09]];
    CONST robtarget point_540_clearance:=[[191,222,149.5],[0,0,1,0],[0, 0, 0, 0],[9E+09,9E+09,9E+09,9E+09,9E+09,9E+09]];
    CONST robtarget point_540_contact:=[[191,222,134.5],[0,0,1,0],[0, 0, 0, 0],[9E+09,9E+09,9E+09,9E+09,9E+09,9E+09]];
    CONST robtarget point_541_contact:=[[191,181,134.5],[0,0,1,0],[0, 0, 0, 0],[9E+09,9E+09,9E+09,9E+09,9E+09,9E+09]];
    CONST robtarget point_541_clearance:=[[191,181,149.5],[0,0,1,0],[0, 0, 0, 0],[9E+09,9E+09,9E+09,9E+09,9E+09,9E+09]];
    CONST robtarget point_542_clearance:=[[308,185,149.5],[0,0,1,0],[0, 0, 0, 0],[9E+09,9E+09,9E+09,9E+09,9E+09,9E+09]];
    CONST robtarget point_542_contact:=[[308,185,134.5],[0,0,1,0],[0, 0, 0, 0],[9E+09,9E+09,9E+09,9E+09,9E+09,9E+09]];
    CONST robtarget point_543_contact:=[[295,187,134.5],[0,0,1,0],[0, 0, 0, 0],[9E+09,9E+09,9E+09,9E+09,9E+09,9E+09]];
    CONST robtarget point_543_clearance:=[[295,187,149.5],[0,0,1,0],[0, 0, 0, 0],[9E+09,9E+09,9E+09,9E+09,9E+09,9E+09]];
    CONST robtarget point_544_clearance:=[[322,186,149.5],[0,0,1,0],[0, 0, 0, 0],[9E+09,9E+09,9E+09,9E+09,9E+09,9E+09]];
    CONST robtarget point_544_contact:=[[322,186,134.5],[0,0,1,0],[0, 0, 0, 0],[9E+09,9E+09,9E+09,9E+09,9E+09,9E+09]];
    CONST robtarget point_545_contact:=[[308,186,134.5],[0,0,1,0],[0, 0, 0, 0],[9E+09,9E+09,9E+09,9E+09,9E+09,9E+09]];
    CONST robtarget point_545_clearance:=[[308,186,149.5],[0,0,1,0],[0, 0, 0, 0],[9E+09,9E+09,9E+09,9E+09,9E+09,9E+09]];
    CONST robtarget point_546_clearance:=[[430,183,149.5],[0,0,1,0],[0, 0, 0, 0],[9E+09,9E+09,9E+09,9E+09,9E+09,9E+09]];
    CONST robtarget point_546_contact:=[[430,183,134.5],[0,0,1,0],[0, 0, 0, 0],[9E+09,9E+09,9E+09,9E+09,9E+09,9E+09]];
    CONST robtarget point_547_contact:=[[423,208,134.5],[0,0,1,0],[0, 0, 0, 0],[9E+09,9E+09,9E+09,9E+09,9E+09,9E+09]];
    CONST robtarget point_547_clearance:=[[423,208,149.5],[0,0,1,0],[0, 0, 0, 0],[9E+09,9E+09,9E+09,9E+09,9E+09,9E+09]];
    CONST robtarget point_548_clearance:=[[296,188,149.5],[0,0,1,0],[0, 0, 0, 0],[9E+09,9E+09,9E+09,9E+09,9E+09,9E+09]];
    CONST robtarget point_548_contact:=[[296,188,134.5],[0,0,1,0],[0, 0, 0, 0],[9E+09,9E+09,9E+09,9E+09,9E+09,9E+09]];
    CONST robtarget point_549_contact:=[[285,184,134.5],[0,0,1,0],[0, 0, 0, 0],[9E+09,9E+09,9E+09,9E+09,9E+09,9E+09]];
    CONST robtarget point_549_clearance:=[[285,184,149.5],[0,0,1,0],[0, 0, 0, 0],[9E+09,9E+09,9E+09,9E+09,9E+09,9E+09]];
    CONST robtarget point_550_clearance:=[[201,186,149.5],[0,0,1,0],[0, 0, 0, 0],[9E+09,9E+09,9E+09,9E+09,9E+09,9E+09]];
    CONST robtarget point_550_contact:=[[201,186,134.5],[0,0,1,0],[0, 0, 0, 0],[9E+09,9E+09,9E+09,9E+09,9E+09,9E+09]];
    CONST robtarget point_551_contact:=[[200,213,134.5],[0,0,1,0],[0, 0, 0, 0],[9E+09,9E+09,9E+09,9E+09,9E+09,9E+09]];
    CONST robtarget point_551_clearance:=[[200,213,149.5],[0,0,1,0],[0, 0, 0, 0],[9E+09,9E+09,9E+09,9E+09,9E+09,9E+09]];
    CONST robtarget point_552_clearance:=[[376,199,149.5],[0,0,1,0],[0, 0, 0, 0],[9E+09,9E+09,9E+09,9E+09,9E+09,9E+09]];
    CONST robtarget point_552_contact:=[[376,199,134.5],[0,0,1,0],[0, 0, 0, 0],[9E+09,9E+09,9E+09,9E+09,9E+09,9E+09]];
    CONST robtarget point_553_contact:=[[381,186,134.5],[0,0,1,0],[0, 0, 0, 0],[9E+09,9E+09,9E+09,9E+09,9E+09,9E+09]];
    CONST robtarget point_553_clearance:=[[381,186,149.5],[0,0,1,0],[0, 0, 0, 0],[9E+09,9E+09,9E+09,9E+09,9E+09,9E+09]];
    CONST robtarget point_554_clearance:=[[376,187,149.5],[0,0,1,0],[0, 0, 0, 0],[9E+09,9E+09,9E+09,9E+09,9E+09,9E+09]];
    CONST robtarget point_554_contact:=[[376,187,134.5],[0,0,1,0],[0, 0, 0, 0],[9E+09,9E+09,9E+09,9E+09,9E+09,9E+09]];
    CONST robtarget point_555_contact:=[[371,210,134.5],[0,0,1,0],[0, 0, 0, 0],[9E+09,9E+09,9E+09,9E+09,9E+09,9E+09]];
    CONST robtarget point_555_clearance:=[[371,210,149.5],[0,0,1,0],[0, 0, 0, 0],[9E+09,9E+09,9E+09,9E+09,9E+09,9E+09]];
    CONST robtarget point_556_clearance:=[[238,191,149.5],[0,0,1,0],[0, 0, 0, 0],[9E+09,9E+09,9E+09,9E+09,9E+09,9E+09]];
    CONST robtarget point_556_contact:=[[238,191,134.5],[0,0,1,0],[0, 0, 0, 0],[9E+09,9E+09,9E+09,9E+09,9E+09,9E+09]];
    CONST robtarget point_557_contact:=[[245,192,134.5],[0,0,1,0],[0, 0, 0, 0],[9E+09,9E+09,9E+09,9E+09,9E+09,9E+09]];
    CONST robtarget point_557_clearance:=[[245,192,149.5],[0,0,1,0],[0, 0, 0, 0],[9E+09,9E+09,9E+09,9E+09,9E+09,9E+09]];
    CONST robtarget point_558_clearance:=[[404,218,149.5],[0,0,1,0],[0, 0, 0, 0],[9E+09,9E+09,9E+09,9E+09,9E+09,9E+09]];
    CONST robtarget point_558_contact:=[[404,218,134.5],[0,0,1,0],[0, 0, 0, 0],[9E+09,9E+09,9E+09,9E+09,9E+09,9E+09]];
    CONST robtarget point_559_contact:=[[413,188,134.5],[0,0,1,0],[0, 0, 0, 0],[9E+09,9E+09,9E+09,9E+09,9E+09,9E+09]];
    CONST robtarget point_559_clearance:=[[413,188,149.5],[0,0,1,0],[0, 0, 0, 0],[9E+09,9E+09,9E+09,9E+09,9E+09,9E+09]];
    CONST robtarget point_560_clearance:=[[226,190,149.5],[0,0,1,0],[0, 0, 0, 0],[9E+09,9E+09,9E+09,9E+09,9E+09,9E+09]];
    CONST robtarget point_560_contact:=[[226,190,134.5],[0,0,1,0],[0, 0, 0, 0],[9E+09,9E+09,9E+09,9E+09,9E+09,9E+09]];
    CONST robtarget point_561_contact:=[[232,197,134.5],[0,0,1,0],[0, 0, 0, 0],[9E+09,9E+09,9E+09,9E+09,9E+09,9E+09]];
    CONST robtarget point_561_clearance:=[[232,197,149.5],[0,0,1,0],[0, 0, 0, 0],[9E+09,9E+09,9E+09,9E+09,9E+09,9E+09]];
    CONST robtarget point_562_clearance:=[[385,191,149.5],[0,0,1,0],[0, 0, 0, 0],[9E+09,9E+09,9E+09,9E+09,9E+09,9E+09]];
    CONST robtarget point_562_contact:=[[385,191,134.5],[0,0,1,0],[0, 0, 0, 0],[9E+09,9E+09,9E+09,9E+09,9E+09,9E+09]];
    CONST robtarget point_563_contact:=[[377,211,134.5],[0,0,1,0],[0, 0, 0, 0],[9E+09,9E+09,9E+09,9E+09,9E+09,9E+09]];
    CONST robtarget point_563_clearance:=[[377,211,149.5],[0,0,1,0],[0, 0, 0, 0],[9E+09,9E+09,9E+09,9E+09,9E+09,9E+09]];
    CONST robtarget point_564_clearance:=[[235,193,149.5],[0,0,1,0],[0, 0, 0, 0],[9E+09,9E+09,9E+09,9E+09,9E+09,9E+09]];
    CONST robtarget point_564_contact:=[[235,193,134.5],[0,0,1,0],[0, 0, 0, 0],[9E+09,9E+09,9E+09,9E+09,9E+09,9E+09]];
    CONST robtarget point_565_contact:=[[253,210,134.5],[0,0,1,0],[0, 0, 0, 0],[9E+09,9E+09,9E+09,9E+09,9E+09,9E+09]];
    CONST robtarget point_565_clearance:=[[253,210,149.5],[0,0,1,0],[0, 0, 0, 0],[9E+09,9E+09,9E+09,9E+09,9E+09,9E+09]];
    CONST robtarget point_566_clearance:=[[397,193,149.5],[0,0,1,0],[0, 0, 0, 0],[9E+09,9E+09,9E+09,9E+09,9E+09,9E+09]];
    CONST robtarget point_566_contact:=[[397,193,134.5],[0,0,1,0],[0, 0, 0, 0],[9E+09,9E+09,9E+09,9E+09,9E+09,9E+09]];
    CONST robtarget point_567_contact:=[[386,220,134.5],[0,0,1,0],[0, 0, 0, 0],[9E+09,9E+09,9E+09,9E+09,9E+09,9E+09]];
    CONST robtarget point_567_clearance:=[[386,220,149.5],[0,0,1,0],[0, 0, 0, 0],[9E+09,9E+09,9E+09,9E+09,9E+09,9E+09]];
    CONST robtarget point_568_clearance:=[[158,197,149.5],[0,0,1,0],[0, 0, 0, 0],[9E+09,9E+09,9E+09,9E+09,9E+09,9E+09]];
    CONST robtarget point_568_contact:=[[158,197,134.5],[0,0,1,0],[0, 0, 0, 0],[9E+09,9E+09,9E+09,9E+09,9E+09,9E+09]];
    CONST robtarget point_569_contact:=[[141,196,134.5],[0,0,1,0],[0, 0, 0, 0],[9E+09,9E+09,9E+09,9E+09,9E+09,9E+09]];
    CONST robtarget point_569_clearance:=[[141,196,149.5],[0,0,1,0],[0, 0, 0, 0],[9E+09,9E+09,9E+09,9E+09,9E+09,9E+09]];
    CONST robtarget point_570_clearance:=[[179,199,149.5],[0,0,1,0],[0, 0, 0, 0],[9E+09,9E+09,9E+09,9E+09,9E+09,9E+09]];
    CONST robtarget point_570_contact:=[[179,199,134.5],[0,0,1,0],[0, 0, 0, 0],[9E+09,9E+09,9E+09,9E+09,9E+09,9E+09]];
    CONST robtarget point_571_contact:=[[165,198,134.5],[0,0,1,0],[0, 0, 0, 0],[9E+09,9E+09,9E+09,9E+09,9E+09,9E+09]];
    CONST robtarget point_571_clearance:=[[165,198,149.5],[0,0,1,0],[0, 0, 0, 0],[9E+09,9E+09,9E+09,9E+09,9E+09,9E+09]];
    CONST robtarget point_572_clearance:=[[180,196,149.5],[0,0,1,0],[0, 0, 0, 0],[9E+09,9E+09,9E+09,9E+09,9E+09,9E+09]];
    CONST robtarget point_572_contact:=[[180,196,134.5],[0,0,1,0],[0, 0, 0, 0],[9E+09,9E+09,9E+09,9E+09,9E+09,9E+09]];
    CONST robtarget point_573_contact:=[[181,201,134.5],[0,0,1,0],[0, 0, 0, 0],[9E+09,9E+09,9E+09,9E+09,9E+09,9E+09]];
    CONST robtarget point_573_clearance:=[[181,201,149.5],[0,0,1,0],[0, 0, 0, 0],[9E+09,9E+09,9E+09,9E+09,9E+09,9E+09]];
    CONST robtarget point_574_clearance:=[[385,205,149.5],[0,0,1,0],[0, 0, 0, 0],[9E+09,9E+09,9E+09,9E+09,9E+09,9E+09]];
    CONST robtarget point_574_contact:=[[385,205,134.5],[0,0,1,0],[0, 0, 0, 0],[9E+09,9E+09,9E+09,9E+09,9E+09,9E+09]];
    CONST robtarget point_575_contact:=[[388,196,134.5],[0,0,1,0],[0, 0, 0, 0],[9E+09,9E+09,9E+09,9E+09,9E+09,9E+09]];
    CONST robtarget point_575_clearance:=[[388,196,149.5],[0,0,1,0],[0, 0, 0, 0],[9E+09,9E+09,9E+09,9E+09,9E+09,9E+09]];
    CONST robtarget point_576_clearance:=[[414,196,149.5],[0,0,1,0],[0, 0, 0, 0],[9E+09,9E+09,9E+09,9E+09,9E+09,9E+09]];
    CONST robtarget point_576_contact:=[[414,196,134.5],[0,0,1,0],[0, 0, 0, 0],[9E+09,9E+09,9E+09,9E+09,9E+09,9E+09]];
    CONST robtarget point_577_contact:=[[411,212,134.5],[0,0,1,0],[0, 0, 0, 0],[9E+09,9E+09,9E+09,9E+09,9E+09,9E+09]];
    CONST robtarget point_577_clearance:=[[411,212,149.5],[0,0,1,0],[0, 0, 0, 0],[9E+09,9E+09,9E+09,9E+09,9E+09,9E+09]];
    CONST robtarget point_578_clearance:=[[406,197,149.5],[0,0,1,0],[0, 0, 0, 0],[9E+09,9E+09,9E+09,9E+09,9E+09,9E+09]];
    CONST robtarget point_578_contact:=[[406,197,134.5],[0,0,1,0],[0, 0, 0, 0],[9E+09,9E+09,9E+09,9E+09,9E+09,9E+09]];
    CONST robtarget point_579_contact:=[[399,219,134.5],[0,0,1,0],[0, 0, 0, 0],[9E+09,9E+09,9E+09,9E+09,9E+09,9E+09]];
    CONST robtarget point_579_clearance:=[[399,219,149.5],[0,0,1,0],[0, 0, 0, 0],[9E+09,9E+09,9E+09,9E+09,9E+09,9E+09]];
    CONST robtarget point_580_clearance:=[[234,215,149.5],[0,0,1,0],[0, 0, 0, 0],[9E+09,9E+09,9E+09,9E+09,9E+09,9E+09]];
    CONST robtarget point_580_contact:=[[234,215,134.5],[0,0,1,0],[0, 0, 0, 0],[9E+09,9E+09,9E+09,9E+09,9E+09,9E+09]];
    CONST robtarget point_581_contact:=[[232,198,134.5],[0,0,1,0],[0, 0, 0, 0],[9E+09,9E+09,9E+09,9E+09,9E+09,9E+09]];
    CONST robtarget point_581_clearance:=[[232,198,149.5],[0,0,1,0],[0, 0, 0, 0],[9E+09,9E+09,9E+09,9E+09,9E+09,9E+09]];
    CONST robtarget point_582_clearance:=[[337,218,149.5],[0,0,1,0],[0, 0, 0, 0],[9E+09,9E+09,9E+09,9E+09,9E+09,9E+09]];
    CONST robtarget point_582_contact:=[[337,218,134.5],[0,0,1,0],[0, 0, 0, 0],[9E+09,9E+09,9E+09,9E+09,9E+09,9E+09]];
    CONST robtarget point_583_contact:=[[358,204,134.5],[0,0,1,0],[0, 0, 0, 0],[9E+09,9E+09,9E+09,9E+09,9E+09,9E+09]];
    CONST robtarget point_583_clearance:=[[358,204,149.5],[0,0,1,0],[0, 0, 0, 0],[9E+09,9E+09,9E+09,9E+09,9E+09,9E+09]];
    CONST robtarget point_584_clearance:=[[184,200,149.5],[0,0,1,0],[0, 0, 0, 0],[9E+09,9E+09,9E+09,9E+09,9E+09,9E+09]];
    CONST robtarget point_584_contact:=[[184,200,134.5],[0,0,1,0],[0, 0, 0, 0],[9E+09,9E+09,9E+09,9E+09,9E+09,9E+09]];
    CONST robtarget point_585_contact:=[[177,204,134.5],[0,0,1,0],[0, 0, 0, 0],[9E+09,9E+09,9E+09,9E+09,9E+09,9E+09]];
    CONST robtarget point_585_clearance:=[[177,204,149.5],[0,0,1,0],[0, 0, 0, 0],[9E+09,9E+09,9E+09,9E+09,9E+09,9E+09]];
    CONST robtarget point_586_clearance:=[[387,227,149.5],[0,0,1,0],[0, 0, 0, 0],[9E+09,9E+09,9E+09,9E+09,9E+09,9E+09]];
    CONST robtarget point_586_contact:=[[387,227,134.5],[0,0,1,0],[0, 0, 0, 0],[9E+09,9E+09,9E+09,9E+09,9E+09,9E+09]];
    CONST robtarget point_587_contact:=[[397,200,134.5],[0,0,1,0],[0, 0, 0, 0],[9E+09,9E+09,9E+09,9E+09,9E+09,9E+09]];
    CONST robtarget point_587_clearance:=[[397,200,149.5],[0,0,1,0],[0, 0, 0, 0],[9E+09,9E+09,9E+09,9E+09,9E+09,9E+09]];
    CONST robtarget point_588_clearance:=[[420,199,149.5],[0,0,1,0],[0, 0, 0, 0],[9E+09,9E+09,9E+09,9E+09,9E+09,9E+09]];
    CONST robtarget point_588_contact:=[[420,199,134.5],[0,0,1,0],[0, 0, 0, 0],[9E+09,9E+09,9E+09,9E+09,9E+09,9E+09]];
    CONST robtarget point_589_contact:=[[417,210,134.5],[0,0,1,0],[0, 0, 0, 0],[9E+09,9E+09,9E+09,9E+09,9E+09,9E+09]];
    CONST robtarget point_589_clearance:=[[417,210,149.5],[0,0,1,0],[0, 0, 0, 0],[9E+09,9E+09,9E+09,9E+09,9E+09,9E+09]];
    CONST robtarget point_590_clearance:=[[431,200,149.5],[0,0,1,0],[0, 0, 0, 0],[9E+09,9E+09,9E+09,9E+09,9E+09,9E+09]];
    CONST robtarget point_590_contact:=[[431,200,134.5],[0,0,1,0],[0, 0, 0, 0],[9E+09,9E+09,9E+09,9E+09,9E+09,9E+09]];
    CONST robtarget point_591_contact:=[[426,215,134.5],[0,0,1,0],[0, 0, 0, 0],[9E+09,9E+09,9E+09,9E+09,9E+09,9E+09]];
    CONST robtarget point_591_clearance:=[[426,215,149.5],[0,0,1,0],[0, 0, 0, 0],[9E+09,9E+09,9E+09,9E+09,9E+09,9E+09]];
    CONST robtarget point_592_clearance:=[[432,212,149.5],[0,0,1,0],[0, 0, 0, 0],[9E+09,9E+09,9E+09,9E+09,9E+09,9E+09]];
    CONST robtarget point_592_contact:=[[432,212,134.5],[0,0,1,0],[0, 0, 0, 0],[9E+09,9E+09,9E+09,9E+09,9E+09,9E+09]];
    CONST robtarget point_593_contact:=[[434,201,134.5],[0,0,1,0],[0, 0, 0, 0],[9E+09,9E+09,9E+09,9E+09,9E+09,9E+09]];
    CONST robtarget point_593_clearance:=[[434,201,149.5],[0,0,1,0],[0, 0, 0, 0],[9E+09,9E+09,9E+09,9E+09,9E+09,9E+09]];
    CONST robtarget point_594_clearance:=[[378,219,149.5],[0,0,1,0],[0, 0, 0, 0],[9E+09,9E+09,9E+09,9E+09,9E+09,9E+09]];
    CONST robtarget point_594_contact:=[[378,219,134.5],[0,0,1,0],[0, 0, 0, 0],[9E+09,9E+09,9E+09,9E+09,9E+09,9E+09]];
    CONST robtarget point_595_contact:=[[387,203,134.5],[0,0,1,0],[0, 0, 0, 0],[9E+09,9E+09,9E+09,9E+09,9E+09,9E+09]];
    CONST robtarget point_595_clearance:=[[387,203,149.5],[0,0,1,0],[0, 0, 0, 0],[9E+09,9E+09,9E+09,9E+09,9E+09,9E+09]];
    CONST robtarget point_596_clearance:=[[422,216,149.5],[0,0,1,0],[0, 0, 0, 0],[9E+09,9E+09,9E+09,9E+09,9E+09,9E+09]];
    CONST robtarget point_596_contact:=[[422,216,134.5],[0,0,1,0],[0, 0, 0, 0],[9E+09,9E+09,9E+09,9E+09,9E+09,9E+09]];
    CONST robtarget point_597_contact:=[[427,203,134.5],[0,0,1,0],[0, 0, 0, 0],[9E+09,9E+09,9E+09,9E+09,9E+09,9E+09]];
    CONST robtarget point_597_clearance:=[[427,203,149.5],[0,0,1,0],[0, 0, 0, 0],[9E+09,9E+09,9E+09,9E+09,9E+09,9E+09]];
    CONST robtarget point_598_clearance:=[[152,205,149.5],[0,0,1,0],[0, 0, 0, 0],[9E+09,9E+09,9E+09,9E+09,9E+09,9E+09]];
    CONST robtarget point_598_contact:=[[152,205,134.5],[0,0,1,0],[0, 0, 0, 0],[9E+09,9E+09,9E+09,9E+09,9E+09,9E+09]];
    CONST robtarget point_599_contact:=[[155,211,134.5],[0,0,1,0],[0, 0, 0, 0],[9E+09,9E+09,9E+09,9E+09,9E+09,9E+09]];
    CONST robtarget point_599_clearance:=[[155,211,149.5],[0,0,1,0],[0, 0, 0, 0],[9E+09,9E+09,9E+09,9E+09,9E+09,9E+09]];
    CONST robtarget point_600_clearance:=[[247,207,149.5],[0,0,1,0],[0, 0, 0, 0],[9E+09,9E+09,9E+09,9E+09,9E+09,9E+09]];
    CONST robtarget point_600_contact:=[[247,207,134.5],[0,0,1,0],[0, 0, 0, 0],[9E+09,9E+09,9E+09,9E+09,9E+09,9E+09]];
    CONST robtarget point_601_contact:=[[245,215,134.5],[0,0,1,0],[0, 0, 0, 0],[9E+09,9E+09,9E+09,9E+09,9E+09,9E+09]];
    CONST robtarget point_601_clearance:=[[245,215,149.5],[0,0,1,0],[0, 0, 0, 0],[9E+09,9E+09,9E+09,9E+09,9E+09,9E+09]];
    CONST robtarget point_602_clearance:=[[268,207,149.5],[0,0,1,0],[0, 0, 0, 0],[9E+09,9E+09,9E+09,9E+09,9E+09,9E+09]];
    CONST robtarget point_602_contact:=[[268,207,134.5],[0,0,1,0],[0, 0, 0, 0],[9E+09,9E+09,9E+09,9E+09,9E+09,9E+09]];
    CONST robtarget point_603_contact:=[[269,214,134.5],[0,0,1,0],[0, 0, 0, 0],[9E+09,9E+09,9E+09,9E+09,9E+09,9E+09]];
    CONST robtarget point_603_clearance:=[[269,214,149.5],[0,0,1,0],[0, 0, 0, 0],[9E+09,9E+09,9E+09,9E+09,9E+09,9E+09]];
    CONST robtarget point_604_clearance:=[[150,208,149.5],[0,0,1,0],[0, 0, 0, 0],[9E+09,9E+09,9E+09,9E+09,9E+09,9E+09]];
    CONST robtarget point_604_contact:=[[150,208,134.5],[0,0,1,0],[0, 0, 0, 0],[9E+09,9E+09,9E+09,9E+09,9E+09,9E+09]];
    CONST robtarget point_605_contact:=[[150,225,134.5],[0,0,1,0],[0, 0, 0, 0],[9E+09,9E+09,9E+09,9E+09,9E+09,9E+09]];
    CONST robtarget point_605_clearance:=[[150,225,149.5],[0,0,1,0],[0, 0, 0, 0],[9E+09,9E+09,9E+09,9E+09,9E+09,9E+09]];
    CONST robtarget point_606_clearance:=[[185,209,149.5],[0,0,1,0],[0, 0, 0, 0],[9E+09,9E+09,9E+09,9E+09,9E+09,9E+09]];
    CONST robtarget point_606_contact:=[[185,209,134.5],[0,0,1,0],[0, 0, 0, 0],[9E+09,9E+09,9E+09,9E+09,9E+09,9E+09]];
    CONST robtarget point_607_contact:=[[175,220,134.5],[0,0,1,0],[0, 0, 0, 0],[9E+09,9E+09,9E+09,9E+09,9E+09,9E+09]];
    CONST robtarget point_607_clearance:=[[175,220,149.5],[0,0,1,0],[0, 0, 0, 0],[9E+09,9E+09,9E+09,9E+09,9E+09,9E+09]];
    CONST robtarget point_608_clearance:=[[204,208,149.5],[0,0,1,0],[0, 0, 0, 0],[9E+09,9E+09,9E+09,9E+09,9E+09,9E+09]];
    CONST robtarget point_608_contact:=[[204,208,134.5],[0,0,1,0],[0, 0, 0, 0],[9E+09,9E+09,9E+09,9E+09,9E+09,9E+09]];
    CONST robtarget point_609_contact:=[[205,218,134.5],[0,0,1,0],[0, 0, 0, 0],[9E+09,9E+09,9E+09,9E+09,9E+09,9E+09]];
    CONST robtarget point_609_clearance:=[[205,218,149.5],[0,0,1,0],[0, 0, 0, 0],[9E+09,9E+09,9E+09,9E+09,9E+09,9E+09]];
    CONST robtarget point_610_clearance:=[[290,209,149.5],[0,0,1,0],[0, 0, 0, 0],[9E+09,9E+09,9E+09,9E+09,9E+09,9E+09]];
    CONST robtarget point_610_contact:=[[290,209,134.5],[0,0,1,0],[0, 0, 0, 0],[9E+09,9E+09,9E+09,9E+09,9E+09,9E+09]];
    CONST robtarget point_611_contact:=[[294,210,134.5],[0,0,1,0],[0, 0, 0, 0],[9E+09,9E+09,9E+09,9E+09,9E+09,9E+09]];
    CONST robtarget point_611_clearance:=[[294,210,149.5],[0,0,1,0],[0, 0, 0, 0],[9E+09,9E+09,9E+09,9E+09,9E+09,9E+09]];
    CONST robtarget point_612_clearance:=[[422,208,149.5],[0,0,1,0],[0, 0, 0, 0],[9E+09,9E+09,9E+09,9E+09,9E+09,9E+09]];
    CONST robtarget point_612_contact:=[[422,208,134.5],[0,0,1,0],[0, 0, 0, 0],[9E+09,9E+09,9E+09,9E+09,9E+09,9E+09]];
    CONST robtarget point_613_contact:=[[417,219,134.5],[0,0,1,0],[0, 0, 0, 0],[9E+09,9E+09,9E+09,9E+09,9E+09,9E+09]];
    CONST robtarget point_613_clearance:=[[417,219,149.5],[0,0,1,0],[0, 0, 0, 0],[9E+09,9E+09,9E+09,9E+09,9E+09,9E+09]];
    CONST robtarget point_614_clearance:=[[161,226,149.5],[0,0,1,0],[0, 0, 0, 0],[9E+09,9E+09,9E+09,9E+09,9E+09,9E+09]];
    CONST robtarget point_614_contact:=[[161,226,134.5],[0,0,1,0],[0, 0, 0, 0],[9E+09,9E+09,9E+09,9E+09,9E+09,9E+09]];
    CONST robtarget point_615_contact:=[[156,210,134.5],[0,0,1,0],[0, 0, 0, 0],[9E+09,9E+09,9E+09,9E+09,9E+09,9E+09]];
    CONST robtarget point_615_clearance:=[[156,210,149.5],[0,0,1,0],[0, 0, 0, 0],[9E+09,9E+09,9E+09,9E+09,9E+09,9E+09]];
    CONST robtarget point_616_clearance:=[[254,210,149.5],[0,0,1,0],[0, 0, 0, 0],[9E+09,9E+09,9E+09,9E+09,9E+09,9E+09]];
    CONST robtarget point_616_contact:=[[254,210,134.5],[0,0,1,0],[0, 0, 0, 0],[9E+09,9E+09,9E+09,9E+09,9E+09,9E+09]];
    CONST robtarget point_617_contact:=[[276,226,134.5],[0,0,1,0],[0, 0, 0, 0],[9E+09,9E+09,9E+09,9E+09,9E+09,9E+09]];
    CONST robtarget point_617_clearance:=[[276,226,149.5],[0,0,1,0],[0, 0, 0, 0],[9E+09,9E+09,9E+09,9E+09,9E+09,9E+09]];
    CONST robtarget point_618_clearance:=[[275,213,149.5],[0,0,1,0],[0, 0, 0, 0],[9E+09,9E+09,9E+09,9E+09,9E+09,9E+09]];
    CONST robtarget point_618_contact:=[[275,213,134.5],[0,0,1,0],[0, 0, 0, 0],[9E+09,9E+09,9E+09,9E+09,9E+09,9E+09]];
    CONST robtarget point_619_contact:=[[283,212,134.5],[0,0,1,0],[0, 0, 0, 0],[9E+09,9E+09,9E+09,9E+09,9E+09,9E+09]];
    CONST robtarget point_619_clearance:=[[283,212,149.5],[0,0,1,0],[0, 0, 0, 0],[9E+09,9E+09,9E+09,9E+09,9E+09,9E+09]];
    CONST robtarget point_620_clearance:=[[294,210,149.5],[0,0,1,0],[0, 0, 0, 0],[9E+09,9E+09,9E+09,9E+09,9E+09,9E+09]];
    CONST robtarget point_620_contact:=[[294,210,134.5],[0,0,1,0],[0, 0, 0, 0],[9E+09,9E+09,9E+09,9E+09,9E+09,9E+09]];
    CONST robtarget point_621_contact:=[[297,212,134.5],[0,0,1,0],[0, 0, 0, 0],[9E+09,9E+09,9E+09,9E+09,9E+09,9E+09]];
    CONST robtarget point_621_clearance:=[[297,212,149.5],[0,0,1,0],[0, 0, 0, 0],[9E+09,9E+09,9E+09,9E+09,9E+09,9E+09]];
    CONST robtarget point_622_clearance:=[[320,215,149.5],[0,0,1,0],[0, 0, 0, 0],[9E+09,9E+09,9E+09,9E+09,9E+09,9E+09]];
    CONST robtarget point_622_contact:=[[320,215,134.5],[0,0,1,0],[0, 0, 0, 0],[9E+09,9E+09,9E+09,9E+09,9E+09,9E+09]];
    CONST robtarget point_623_contact:=[[326,210,134.5],[0,0,1,0],[0, 0, 0, 0],[9E+09,9E+09,9E+09,9E+09,9E+09,9E+09]];
    CONST robtarget point_623_clearance:=[[326,210,149.5],[0,0,1,0],[0, 0, 0, 0],[9E+09,9E+09,9E+09,9E+09,9E+09,9E+09]];
    CONST robtarget point_624_clearance:=[[167,210,149.5],[0,0,1,0],[0, 0, 0, 0],[9E+09,9E+09,9E+09,9E+09,9E+09,9E+09]];
    CONST robtarget point_624_contact:=[[167,210,134.5],[0,0,1,0],[0, 0, 0, 0],[9E+09,9E+09,9E+09,9E+09,9E+09,9E+09]];
    CONST robtarget point_625_contact:=[[170,217,134.5],[0,0,1,0],[0, 0, 0, 0],[9E+09,9E+09,9E+09,9E+09,9E+09,9E+09]];
    CONST robtarget point_625_clearance:=[[170,217,149.5],[0,0,1,0],[0, 0, 0, 0],[9E+09,9E+09,9E+09,9E+09,9E+09,9E+09]];
    CONST robtarget point_626_clearance:=[[169,216,149.5],[0,0,1,0],[0, 0, 0, 0],[9E+09,9E+09,9E+09,9E+09,9E+09,9E+09]];
    CONST robtarget point_626_contact:=[[169,216,134.5],[0,0,1,0],[0, 0, 0, 0],[9E+09,9E+09,9E+09,9E+09,9E+09,9E+09]];
    CONST robtarget point_627_contact:=[[176,212,134.5],[0,0,1,0],[0, 0, 0, 0],[9E+09,9E+09,9E+09,9E+09,9E+09,9E+09]];
    CONST robtarget point_627_clearance:=[[176,212,149.5],[0,0,1,0],[0, 0, 0, 0],[9E+09,9E+09,9E+09,9E+09,9E+09,9E+09]];
    CONST robtarget point_628_clearance:=[[208,211,149.5],[0,0,1,0],[0, 0, 0, 0],[9E+09,9E+09,9E+09,9E+09,9E+09,9E+09]];
    CONST robtarget point_628_contact:=[[208,211,134.5],[0,0,1,0],[0, 0, 0, 0],[9E+09,9E+09,9E+09,9E+09,9E+09,9E+09]];
    CONST robtarget point_629_contact:=[[213,239,134.5],[0,0,1,0],[0, 0, 0, 0],[9E+09,9E+09,9E+09,9E+09,9E+09,9E+09]];
    CONST robtarget point_629_clearance:=[[213,239,149.5],[0,0,1,0],[0, 0, 0, 0],[9E+09,9E+09,9E+09,9E+09,9E+09,9E+09]];
    CONST robtarget point_630_clearance:=[[267,218,149.5],[0,0,1,0],[0, 0, 0, 0],[9E+09,9E+09,9E+09,9E+09,9E+09,9E+09]];
    CONST robtarget point_630_contact:=[[267,218,134.5],[0,0,1,0],[0, 0, 0, 0],[9E+09,9E+09,9E+09,9E+09,9E+09,9E+09]];
    CONST robtarget point_631_contact:=[[337,219,134.5],[0,0,1,0],[0, 0, 0, 0],[9E+09,9E+09,9E+09,9E+09,9E+09,9E+09]];
    CONST robtarget point_631_clearance:=[[337,219,149.5],[0,0,1,0],[0, 0, 0, 0],[9E+09,9E+09,9E+09,9E+09,9E+09,9E+09]];
    CONST robtarget point_632_clearance:=[[376,212,149.5],[0,0,1,0],[0, 0, 0, 0],[9E+09,9E+09,9E+09,9E+09,9E+09,9E+09]];
    CONST robtarget point_632_contact:=[[376,212,134.5],[0,0,1,0],[0, 0, 0, 0],[9E+09,9E+09,9E+09,9E+09,9E+09,9E+09]];
    CONST robtarget point_633_contact:=[[373,218,134.5],[0,0,1,0],[0, 0, 0, 0],[9E+09,9E+09,9E+09,9E+09,9E+09,9E+09]];
    CONST robtarget point_633_clearance:=[[373,218,149.5],[0,0,1,0],[0, 0, 0, 0],[9E+09,9E+09,9E+09,9E+09,9E+09,9E+09]];
    CONST robtarget point_634_clearance:=[[234,240,149.5],[0,0,1,0],[0, 0, 0, 0],[9E+09,9E+09,9E+09,9E+09,9E+09,9E+09]];
    CONST robtarget point_634_contact:=[[234,240,134.5],[0,0,1,0],[0, 0, 0, 0],[9E+09,9E+09,9E+09,9E+09,9E+09,9E+09]];
    CONST robtarget point_635_contact:=[[236,213,134.5],[0,0,1,0],[0, 0, 0, 0],[9E+09,9E+09,9E+09,9E+09,9E+09,9E+09]];
    CONST robtarget point_635_clearance:=[[236,213,149.5],[0,0,1,0],[0, 0, 0, 0],[9E+09,9E+09,9E+09,9E+09,9E+09,9E+09]];
    CONST robtarget point_636_clearance:=[[410,213,149.5],[0,0,1,0],[0, 0, 0, 0],[9E+09,9E+09,9E+09,9E+09,9E+09,9E+09]];
    CONST robtarget point_636_contact:=[[410,213,134.5],[0,0,1,0],[0, 0, 0, 0],[9E+09,9E+09,9E+09,9E+09,9E+09,9E+09]];
    CONST robtarget point_637_contact:=[[410,218,134.5],[0,0,1,0],[0, 0, 0, 0],[9E+09,9E+09,9E+09,9E+09,9E+09,9E+09]];
    CONST robtarget point_637_clearance:=[[410,218,149.5],[0,0,1,0],[0, 0, 0, 0],[9E+09,9E+09,9E+09,9E+09,9E+09,9E+09]];
    CONST robtarget point_638_clearance:=[[434,220,149.5],[0,0,1,0],[0, 0, 0, 0],[9E+09,9E+09,9E+09,9E+09,9E+09,9E+09]];
    CONST robtarget point_638_contact:=[[434,220,134.5],[0,0,1,0],[0, 0, 0, 0],[9E+09,9E+09,9E+09,9E+09,9E+09,9E+09]];
    CONST robtarget point_639_contact:=[[427,215,134.5],[0,0,1,0],[0, 0, 0, 0],[9E+09,9E+09,9E+09,9E+09,9E+09,9E+09]];
    CONST robtarget point_639_clearance:=[[427,215,149.5],[0,0,1,0],[0, 0, 0, 0],[9E+09,9E+09,9E+09,9E+09,9E+09,9E+09]];
    CONST robtarget point_640_clearance:=[[139,215,149.5],[0,0,1,0],[0, 0, 0, 0],[9E+09,9E+09,9E+09,9E+09,9E+09,9E+09]];
    CONST robtarget point_640_contact:=[[139,215,134.5],[0,0,1,0],[0, 0, 0, 0],[9E+09,9E+09,9E+09,9E+09,9E+09,9E+09]];
    CONST robtarget point_641_contact:=[[147,220,134.5],[0,0,1,0],[0, 0, 0, 0],[9E+09,9E+09,9E+09,9E+09,9E+09,9E+09]];
    CONST robtarget point_641_clearance:=[[147,220,149.5],[0,0,1,0],[0, 0, 0, 0],[9E+09,9E+09,9E+09,9E+09,9E+09,9E+09]];
    CONST robtarget point_642_clearance:=[[200,214,149.5],[0,0,1,0],[0, 0, 0, 0],[9E+09,9E+09,9E+09,9E+09,9E+09,9E+09]];
    CONST robtarget point_642_contact:=[[200,214,134.5],[0,0,1,0],[0, 0, 0, 0],[9E+09,9E+09,9E+09,9E+09,9E+09,9E+09]];
    CONST robtarget point_643_contact:=[[203,230,134.5],[0,0,1,0],[0, 0, 0, 0],[9E+09,9E+09,9E+09,9E+09,9E+09,9E+09]];
    CONST robtarget point_643_clearance:=[[203,230,149.5],[0,0,1,0],[0, 0, 0, 0],[9E+09,9E+09,9E+09,9E+09,9E+09,9E+09]];
    CONST robtarget point_644_clearance:=[[257,220,149.5],[0,0,1,0],[0, 0, 0, 0],[9E+09,9E+09,9E+09,9E+09,9E+09,9E+09]];
    CONST robtarget point_644_contact:=[[257,220,134.5],[0,0,1,0],[0, 0, 0, 0],[9E+09,9E+09,9E+09,9E+09,9E+09,9E+09]];
    CONST robtarget point_645_contact:=[[254,215,134.5],[0,0,1,0],[0, 0, 0, 0],[9E+09,9E+09,9E+09,9E+09,9E+09,9E+09]];
    CONST robtarget point_645_clearance:=[[254,215,149.5],[0,0,1,0],[0, 0, 0, 0],[9E+09,9E+09,9E+09,9E+09,9E+09,9E+09]];
    CONST robtarget point_646_clearance:=[[343,224,149.5],[0,0,1,0],[0, 0, 0, 0],[9E+09,9E+09,9E+09,9E+09,9E+09,9E+09]];
    CONST robtarget point_646_contact:=[[343,224,134.5],[0,0,1,0],[0, 0, 0, 0],[9E+09,9E+09,9E+09,9E+09,9E+09,9E+09]];
    CONST robtarget point_647_contact:=[[349,214,134.5],[0,0,1,0],[0, 0, 0, 0],[9E+09,9E+09,9E+09,9E+09,9E+09,9E+09]];
    CONST robtarget point_647_clearance:=[[349,214,149.5],[0,0,1,0],[0, 0, 0, 0],[9E+09,9E+09,9E+09,9E+09,9E+09,9E+09]];
    CONST robtarget point_648_clearance:=[[412,214,149.5],[0,0,1,0],[0, 0, 0, 0],[9E+09,9E+09,9E+09,9E+09,9E+09,9E+09]];
    CONST robtarget point_648_contact:=[[412,214,134.5],[0,0,1,0],[0, 0, 0, 0],[9E+09,9E+09,9E+09,9E+09,9E+09,9E+09]];
    CONST robtarget point_649_contact:=[[416,221,134.5],[0,0,1,0],[0, 0, 0, 0],[9E+09,9E+09,9E+09,9E+09,9E+09,9E+09]];
    CONST robtarget point_649_clearance:=[[416,221,149.5],[0,0,1,0],[0, 0, 0, 0],[9E+09,9E+09,9E+09,9E+09,9E+09,9E+09]];
    CONST robtarget point_650_clearance:=[[245,216,149.5],[0,0,1,0],[0, 0, 0, 0],[9E+09,9E+09,9E+09,9E+09,9E+09,9E+09]];
    CONST robtarget point_650_contact:=[[245,216,134.5],[0,0,1,0],[0, 0, 0, 0],[9E+09,9E+09,9E+09,9E+09,9E+09,9E+09]];
    CONST robtarget point_651_contact:=[[245,222,134.5],[0,0,1,0],[0, 0, 0, 0],[9E+09,9E+09,9E+09,9E+09,9E+09,9E+09]];
    CONST robtarget point_651_clearance:=[[245,222,149.5],[0,0,1,0],[0, 0, 0, 0],[9E+09,9E+09,9E+09,9E+09,9E+09,9E+09]];
    CONST robtarget point_652_clearance:=[[251,216,149.5],[0,0,1,0],[0, 0, 0, 0],[9E+09,9E+09,9E+09,9E+09,9E+09,9E+09]];
    CONST robtarget point_652_contact:=[[251,216,134.5],[0,0,1,0],[0, 0, 0, 0],[9E+09,9E+09,9E+09,9E+09,9E+09,9E+09]];
    CONST robtarget point_653_contact:=[[252,216,134.5],[0,0,1,0],[0, 0, 0, 0],[9E+09,9E+09,9E+09,9E+09,9E+09,9E+09]];
    CONST robtarget point_653_clearance:=[[252,216,149.5],[0,0,1,0],[0, 0, 0, 0],[9E+09,9E+09,9E+09,9E+09,9E+09,9E+09]];
    CONST robtarget point_654_clearance:=[[183,217,149.5],[0,0,1,0],[0, 0, 0, 0],[9E+09,9E+09,9E+09,9E+09,9E+09,9E+09]];
    CONST robtarget point_654_contact:=[[183,217,134.5],[0,0,1,0],[0, 0, 0, 0],[9E+09,9E+09,9E+09,9E+09,9E+09,9E+09]];
    CONST robtarget point_655_contact:=[[181,226,134.5],[0,0,1,0],[0, 0, 0, 0],[9E+09,9E+09,9E+09,9E+09,9E+09,9E+09]];
    CONST robtarget point_655_clearance:=[[181,226,149.5],[0,0,1,0],[0, 0, 0, 0],[9E+09,9E+09,9E+09,9E+09,9E+09,9E+09]];
    CONST robtarget point_656_clearance:=[[252,217,149.5],[0,0,1,0],[0, 0, 0, 0],[9E+09,9E+09,9E+09,9E+09,9E+09,9E+09]];
    CONST robtarget point_656_contact:=[[252,217,134.5],[0,0,1,0],[0, 0, 0, 0],[9E+09,9E+09,9E+09,9E+09,9E+09,9E+09]];
    CONST robtarget point_657_contact:=[[253,223,134.5],[0,0,1,0],[0, 0, 0, 0],[9E+09,9E+09,9E+09,9E+09,9E+09,9E+09]];
    CONST robtarget point_657_clearance:=[[253,223,149.5],[0,0,1,0],[0, 0, 0, 0],[9E+09,9E+09,9E+09,9E+09,9E+09,9E+09]];
    CONST robtarget point_658_clearance:=[[261,251,149.5],[0,0,1,0],[0, 0, 0, 0],[9E+09,9E+09,9E+09,9E+09,9E+09,9E+09]];
    CONST robtarget point_658_contact:=[[261,251,134.5],[0,0,1,0],[0, 0, 0, 0],[9E+09,9E+09,9E+09,9E+09,9E+09,9E+09]];
    CONST robtarget point_659_contact:=[[257,219,134.5],[0,0,1,0],[0, 0, 0, 0],[9E+09,9E+09,9E+09,9E+09,9E+09,9E+09]];
    CONST robtarget point_659_clearance:=[[257,219,149.5],[0,0,1,0],[0, 0, 0, 0],[9E+09,9E+09,9E+09,9E+09,9E+09,9E+09]];
    CONST robtarget point_660_clearance:=[[180,220,149.5],[0,0,1,0],[0, 0, 0, 0],[9E+09,9E+09,9E+09,9E+09,9E+09,9E+09]];
    CONST robtarget point_660_contact:=[[180,220,134.5],[0,0,1,0],[0, 0, 0, 0],[9E+09,9E+09,9E+09,9E+09,9E+09,9E+09]];
    CONST robtarget point_661_contact:=[[176,226,134.5],[0,0,1,0],[0, 0, 0, 0],[9E+09,9E+09,9E+09,9E+09,9E+09,9E+09]];
    CONST robtarget point_661_clearance:=[[176,226,149.5],[0,0,1,0],[0, 0, 0, 0],[9E+09,9E+09,9E+09,9E+09,9E+09,9E+09]];
    CONST robtarget point_662_clearance:=[[387,221,149.5],[0,0,1,0],[0, 0, 0, 0],[9E+09,9E+09,9E+09,9E+09,9E+09,9E+09]];
    CONST robtarget point_662_contact:=[[387,221,134.5],[0,0,1,0],[0, 0, 0, 0],[9E+09,9E+09,9E+09,9E+09,9E+09,9E+09]];
    CONST robtarget point_663_contact:=[[380,225,134.5],[0,0,1,0],[0, 0, 0, 0],[9E+09,9E+09,9E+09,9E+09,9E+09,9E+09]];
    CONST robtarget point_663_clearance:=[[380,225,149.5],[0,0,1,0],[0, 0, 0, 0],[9E+09,9E+09,9E+09,9E+09,9E+09,9E+09]];
    CONST robtarget point_664_clearance:=[[412,220,149.5],[0,0,1,0],[0, 0, 0, 0],[9E+09,9E+09,9E+09,9E+09,9E+09,9E+09]];
    CONST robtarget point_664_contact:=[[412,220,134.5],[0,0,1,0],[0, 0, 0, 0],[9E+09,9E+09,9E+09,9E+09,9E+09,9E+09]];
    CONST robtarget point_665_contact:=[[411,230,134.5],[0,0,1,0],[0, 0, 0, 0],[9E+09,9E+09,9E+09,9E+09,9E+09,9E+09]];
    CONST robtarget point_665_clearance:=[[411,230,149.5],[0,0,1,0],[0, 0, 0, 0],[9E+09,9E+09,9E+09,9E+09,9E+09,9E+09]];
    CONST robtarget point_666_clearance:=[[146,223,149.5],[0,0,1,0],[0, 0, 0, 0],[9E+09,9E+09,9E+09,9E+09,9E+09,9E+09]];
    CONST robtarget point_666_contact:=[[146,223,134.5],[0,0,1,0],[0, 0, 0, 0],[9E+09,9E+09,9E+09,9E+09,9E+09,9E+09]];
    CONST robtarget point_667_contact:=[[138,222,134.5],[0,0,1,0],[0, 0, 0, 0],[9E+09,9E+09,9E+09,9E+09,9E+09,9E+09]];
    CONST robtarget point_667_clearance:=[[138,222,149.5],[0,0,1,0],[0, 0, 0, 0],[9E+09,9E+09,9E+09,9E+09,9E+09,9E+09]];
    CONST robtarget point_668_clearance:=[[185,235,149.5],[0,0,1,0],[0, 0, 0, 0],[9E+09,9E+09,9E+09,9E+09,9E+09,9E+09]];
    CONST robtarget point_668_contact:=[[185,235,134.5],[0,0,1,0],[0, 0, 0, 0],[9E+09,9E+09,9E+09,9E+09,9E+09,9E+09]];
    CONST robtarget point_669_contact:=[[187,223,134.5],[0,0,1,0],[0, 0, 0, 0],[9E+09,9E+09,9E+09,9E+09,9E+09,9E+09]];
    CONST robtarget point_669_clearance:=[[187,223,149.5],[0,0,1,0],[0, 0, 0, 0],[9E+09,9E+09,9E+09,9E+09,9E+09,9E+09]];
    CONST robtarget point_670_clearance:=[[197,237,149.5],[0,0,1,0],[0, 0, 0, 0],[9E+09,9E+09,9E+09,9E+09,9E+09,9E+09]];
    CONST robtarget point_670_contact:=[[197,237,134.5],[0,0,1,0],[0, 0, 0, 0],[9E+09,9E+09,9E+09,9E+09,9E+09,9E+09]];
    CONST robtarget point_671_contact:=[[195,223,134.5],[0,0,1,0],[0, 0, 0, 0],[9E+09,9E+09,9E+09,9E+09,9E+09,9E+09]];
    CONST robtarget point_671_clearance:=[[195,223,149.5],[0,0,1,0],[0, 0, 0, 0],[9E+09,9E+09,9E+09,9E+09,9E+09,9E+09]];
    CONST robtarget point_672_clearance:=[[245,223,149.5],[0,0,1,0],[0, 0, 0, 0],[9E+09,9E+09,9E+09,9E+09,9E+09,9E+09]];
    CONST robtarget point_672_contact:=[[245,223,134.5],[0,0,1,0],[0, 0, 0, 0],[9E+09,9E+09,9E+09,9E+09,9E+09,9E+09]];
    CONST robtarget point_673_contact:=[[246,231,134.5],[0,0,1,0],[0, 0, 0, 0],[9E+09,9E+09,9E+09,9E+09,9E+09,9E+09]];
    CONST robtarget point_673_clearance:=[[246,231,149.5],[0,0,1,0],[0, 0, 0, 0],[9E+09,9E+09,9E+09,9E+09,9E+09,9E+09]];
    CONST robtarget point_674_clearance:=[[138,227,149.5],[0,0,1,0],[0, 0, 0, 0],[9E+09,9E+09,9E+09,9E+09,9E+09,9E+09]];
    CONST robtarget point_674_contact:=[[138,227,134.5],[0,0,1,0],[0, 0, 0, 0],[9E+09,9E+09,9E+09,9E+09,9E+09,9E+09]];
    CONST robtarget point_675_contact:=[[163,227,134.5],[0,0,1,0],[0, 0, 0, 0],[9E+09,9E+09,9E+09,9E+09,9E+09,9E+09]];
    CONST robtarget point_675_clearance:=[[163,227,149.5],[0,0,1,0],[0, 0, 0, 0],[9E+09,9E+09,9E+09,9E+09,9E+09,9E+09]];
    CONST robtarget point_676_clearance:=[[253,225,149.5],[0,0,1,0],[0, 0, 0, 0],[9E+09,9E+09,9E+09,9E+09,9E+09,9E+09]];
    CONST robtarget point_676_contact:=[[253,225,134.5],[0,0,1,0],[0, 0, 0, 0],[9E+09,9E+09,9E+09,9E+09,9E+09,9E+09]];
    CONST robtarget point_677_contact:=[[253,230,134.5],[0,0,1,0],[0, 0, 0, 0],[9E+09,9E+09,9E+09,9E+09,9E+09,9E+09]];
    CONST robtarget point_677_clearance:=[[253,230,149.5],[0,0,1,0],[0, 0, 0, 0],[9E+09,9E+09,9E+09,9E+09,9E+09,9E+09]];
    CONST robtarget point_678_clearance:=[[327,226,149.5],[0,0,1,0],[0, 0, 0, 0],[9E+09,9E+09,9E+09,9E+09,9E+09,9E+09]];
    CONST robtarget point_678_contact:=[[327,226,134.5],[0,0,1,0],[0, 0, 0, 0],[9E+09,9E+09,9E+09,9E+09,9E+09,9E+09]];
    CONST robtarget point_679_contact:=[[298,229,134.5],[0,0,1,0],[0, 0, 0, 0],[9E+09,9E+09,9E+09,9E+09,9E+09,9E+09]];
    CONST robtarget point_679_clearance:=[[298,229,149.5],[0,0,1,0],[0, 0, 0, 0],[9E+09,9E+09,9E+09,9E+09,9E+09,9E+09]];
    CONST robtarget point_680_clearance:=[[344,225,149.5],[0,0,1,0],[0, 0, 0, 0],[9E+09,9E+09,9E+09,9E+09,9E+09,9E+09]];
    CONST robtarget point_680_contact:=[[344,225,134.5],[0,0,1,0],[0, 0, 0, 0],[9E+09,9E+09,9E+09,9E+09,9E+09,9E+09]];
    CONST robtarget point_681_contact:=[[349,235,134.5],[0,0,1,0],[0, 0, 0, 0],[9E+09,9E+09,9E+09,9E+09,9E+09,9E+09]];
    CONST robtarget point_681_clearance:=[[349,235,149.5],[0,0,1,0],[0, 0, 0, 0],[9E+09,9E+09,9E+09,9E+09,9E+09,9E+09]];
    CONST robtarget point_682_clearance:=[[325,236,149.5],[0,0,1,0],[0, 0, 0, 0],[9E+09,9E+09,9E+09,9E+09,9E+09,9E+09]];
    CONST robtarget point_682_contact:=[[325,236,134.5],[0,0,1,0],[0, 0, 0, 0],[9E+09,9E+09,9E+09,9E+09,9E+09,9E+09]];
    CONST robtarget point_683_contact:=[[327,227,134.5],[0,0,1,0],[0, 0, 0, 0],[9E+09,9E+09,9E+09,9E+09,9E+09,9E+09]];
    CONST robtarget point_683_clearance:=[[327,227,149.5],[0,0,1,0],[0, 0, 0, 0],[9E+09,9E+09,9E+09,9E+09,9E+09,9E+09]];
    CONST robtarget point_684_clearance:=[[157,237,149.5],[0,0,1,0],[0, 0, 0, 0],[9E+09,9E+09,9E+09,9E+09,9E+09,9E+09]];
    CONST robtarget point_684_contact:=[[157,237,134.5],[0,0,1,0],[0, 0, 0, 0],[9E+09,9E+09,9E+09,9E+09,9E+09,9E+09]];
    CONST robtarget point_685_contact:=[[171,229,134.5],[0,0,1,0],[0, 0, 0, 0],[9E+09,9E+09,9E+09,9E+09,9E+09,9E+09]];
    CONST robtarget point_685_clearance:=[[171,229,149.5],[0,0,1,0],[0, 0, 0, 0],[9E+09,9E+09,9E+09,9E+09,9E+09,9E+09]];
    CONST robtarget point_686_clearance:=[[178,228,149.5],[0,0,1,0],[0, 0, 0, 0],[9E+09,9E+09,9E+09,9E+09,9E+09,9E+09]];
    CONST robtarget point_686_contact:=[[178,228,134.5],[0,0,1,0],[0, 0, 0, 0],[9E+09,9E+09,9E+09,9E+09,9E+09,9E+09]];
    CONST robtarget point_687_contact:=[[178,232,134.5],[0,0,1,0],[0, 0, 0, 0],[9E+09,9E+09,9E+09,9E+09,9E+09,9E+09]];
    CONST robtarget point_687_clearance:=[[178,232,149.5],[0,0,1,0],[0, 0, 0, 0],[9E+09,9E+09,9E+09,9E+09,9E+09,9E+09]];
    CONST robtarget point_688_clearance:=[[182,228,149.5],[0,0,1,0],[0, 0, 0, 0],[9E+09,9E+09,9E+09,9E+09,9E+09,9E+09]];
    CONST robtarget point_688_contact:=[[182,228,134.5],[0,0,1,0],[0, 0, 0, 0],[9E+09,9E+09,9E+09,9E+09,9E+09,9E+09]];
    CONST robtarget point_689_contact:=[[181,234,134.5],[0,0,1,0],[0, 0, 0, 0],[9E+09,9E+09,9E+09,9E+09,9E+09,9E+09]];
    CONST robtarget point_689_clearance:=[[181,234,149.5],[0,0,1,0],[0, 0, 0, 0],[9E+09,9E+09,9E+09,9E+09,9E+09,9E+09]];
    CONST robtarget point_690_clearance:=[[410,229,149.5],[0,0,1,0],[0, 0, 0, 0],[9E+09,9E+09,9E+09,9E+09,9E+09,9E+09]];
    CONST robtarget point_690_contact:=[[410,229,134.5],[0,0,1,0],[0, 0, 0, 0],[9E+09,9E+09,9E+09,9E+09,9E+09,9E+09]];
    CONST robtarget point_691_contact:=[[401,240,134.5],[0,0,1,0],[0, 0, 0, 0],[9E+09,9E+09,9E+09,9E+09,9E+09,9E+09]];
    CONST robtarget point_691_clearance:=[[401,240,149.5],[0,0,1,0],[0, 0, 0, 0],[9E+09,9E+09,9E+09,9E+09,9E+09,9E+09]];
    CONST robtarget point_692_clearance:=[[417,230,149.5],[0,0,1,0],[0, 0, 0, 0],[9E+09,9E+09,9E+09,9E+09,9E+09,9E+09]];
    CONST robtarget point_692_contact:=[[417,230,134.5],[0,0,1,0],[0, 0, 0, 0],[9E+09,9E+09,9E+09,9E+09,9E+09,9E+09]];
    CONST robtarget point_693_contact:=[[412,236,134.5],[0,0,1,0],[0, 0, 0, 0],[9E+09,9E+09,9E+09,9E+09,9E+09,9E+09]];
    CONST robtarget point_693_clearance:=[[412,236,149.5],[0,0,1,0],[0, 0, 0, 0],[9E+09,9E+09,9E+09,9E+09,9E+09,9E+09]];
    CONST robtarget point_694_clearance:=[[191,246,149.5],[0,0,1,0],[0, 0, 0, 0],[9E+09,9E+09,9E+09,9E+09,9E+09,9E+09]];
    CONST robtarget point_694_contact:=[[191,246,134.5],[0,0,1,0],[0, 0, 0, 0],[9E+09,9E+09,9E+09,9E+09,9E+09,9E+09]];
    CONST robtarget point_695_contact:=[[194,231,134.5],[0,0,1,0],[0, 0, 0, 0],[9E+09,9E+09,9E+09,9E+09,9E+09,9E+09]];
    CONST robtarget point_695_clearance:=[[194,231,149.5],[0,0,1,0],[0, 0, 0, 0],[9E+09,9E+09,9E+09,9E+09,9E+09,9E+09]];
    CONST robtarget point_696_clearance:=[[247,231,149.5],[0,0,1,0],[0, 0, 0, 0],[9E+09,9E+09,9E+09,9E+09,9E+09,9E+09]];
    CONST robtarget point_696_contact:=[[247,231,134.5],[0,0,1,0],[0, 0, 0, 0],[9E+09,9E+09,9E+09,9E+09,9E+09,9E+09]];
    CONST robtarget point_697_contact:=[[258,252,134.5],[0,0,1,0],[0, 0, 0, 0],[9E+09,9E+09,9E+09,9E+09,9E+09,9E+09]];
    CONST robtarget point_697_clearance:=[[258,252,149.5],[0,0,1,0],[0, 0, 0, 0],[9E+09,9E+09,9E+09,9E+09,9E+09,9E+09]];
    CONST robtarget point_698_clearance:=[[252,231,149.5],[0,0,1,0],[0, 0, 0, 0],[9E+09,9E+09,9E+09,9E+09,9E+09,9E+09]];
    CONST robtarget point_698_contact:=[[252,231,134.5],[0,0,1,0],[0, 0, 0, 0],[9E+09,9E+09,9E+09,9E+09,9E+09,9E+09]];
    CONST robtarget point_699_contact:=[[255,239,134.5],[0,0,1,0],[0, 0, 0, 0],[9E+09,9E+09,9E+09,9E+09,9E+09,9E+09]];
    CONST robtarget point_699_clearance:=[[255,239,149.5],[0,0,1,0],[0, 0, 0, 0],[9E+09,9E+09,9E+09,9E+09,9E+09,9E+09]];
    CONST robtarget point_700_clearance:=[[319,231,149.5],[0,0,1,0],[0, 0, 0, 0],[9E+09,9E+09,9E+09,9E+09,9E+09,9E+09]];
    CONST robtarget point_700_contact:=[[319,231,134.5],[0,0,1,0],[0, 0, 0, 0],[9E+09,9E+09,9E+09,9E+09,9E+09,9E+09]];
    CONST robtarget point_701_contact:=[[312,233,134.5],[0,0,1,0],[0, 0, 0, 0],[9E+09,9E+09,9E+09,9E+09,9E+09,9E+09]];
    CONST robtarget point_701_clearance:=[[312,233,149.5],[0,0,1,0],[0, 0, 0, 0],[9E+09,9E+09,9E+09,9E+09,9E+09,9E+09]];
    CONST robtarget point_702_clearance:=[[384,232,149.5],[0,0,1,0],[0, 0, 0, 0],[9E+09,9E+09,9E+09,9E+09,9E+09,9E+09]];
    CONST robtarget point_702_contact:=[[384,232,134.5],[0,0,1,0],[0, 0, 0, 0],[9E+09,9E+09,9E+09,9E+09,9E+09,9E+09]];
    CONST robtarget point_703_contact:=[[371,245,134.5],[0,0,1,0],[0, 0, 0, 0],[9E+09,9E+09,9E+09,9E+09,9E+09,9E+09]];
    CONST robtarget point_703_clearance:=[[371,245,149.5],[0,0,1,0],[0, 0, 0, 0],[9E+09,9E+09,9E+09,9E+09,9E+09,9E+09]];
    CONST robtarget point_704_clearance:=[[202,250,149.5],[0,0,1,0],[0, 0, 0, 0],[9E+09,9E+09,9E+09,9E+09,9E+09,9E+09]];
    CONST robtarget point_704_contact:=[[202,250,134.5],[0,0,1,0],[0, 0, 0, 0],[9E+09,9E+09,9E+09,9E+09,9E+09,9E+09]];
    CONST robtarget point_705_contact:=[[198,232,134.5],[0,0,1,0],[0, 0, 0, 0],[9E+09,9E+09,9E+09,9E+09,9E+09,9E+09]];
    CONST robtarget point_705_clearance:=[[198,232,149.5],[0,0,1,0],[0, 0, 0, 0],[9E+09,9E+09,9E+09,9E+09,9E+09,9E+09]];
    CONST robtarget point_706_clearance:=[[377,250,149.5],[0,0,1,0],[0, 0, 0, 0],[9E+09,9E+09,9E+09,9E+09,9E+09,9E+09]];
    CONST robtarget point_706_contact:=[[377,250,134.5],[0,0,1,0],[0, 0, 0, 0],[9E+09,9E+09,9E+09,9E+09,9E+09,9E+09]];
    CONST robtarget point_707_contact:=[[392,232,134.5],[0,0,1,0],[0, 0, 0, 0],[9E+09,9E+09,9E+09,9E+09,9E+09,9E+09]];
    CONST robtarget point_707_clearance:=[[392,232,149.5],[0,0,1,0],[0, 0, 0, 0],[9E+09,9E+09,9E+09,9E+09,9E+09,9E+09]];
    CONST robtarget point_708_clearance:=[[397,233,149.5],[0,0,1,0],[0, 0, 0, 0],[9E+09,9E+09,9E+09,9E+09,9E+09,9E+09]];
    CONST robtarget point_708_contact:=[[397,233,134.5],[0,0,1,0],[0, 0, 0, 0],[9E+09,9E+09,9E+09,9E+09,9E+09,9E+09]];
    CONST robtarget point_709_contact:=[[383,250,134.5],[0,0,1,0],[0, 0, 0, 0],[9E+09,9E+09,9E+09,9E+09,9E+09,9E+09]];
    CONST robtarget point_709_clearance:=[[383,250,149.5],[0,0,1,0],[0, 0, 0, 0],[9E+09,9E+09,9E+09,9E+09,9E+09,9E+09]];
    CONST robtarget point_710_clearance:=[[223,243,149.5],[0,0,1,0],[0, 0, 0, 0],[9E+09,9E+09,9E+09,9E+09,9E+09,9E+09]];
    CONST robtarget point_710_contact:=[[223,243,134.5],[0,0,1,0],[0, 0, 0, 0],[9E+09,9E+09,9E+09,9E+09,9E+09,9E+09]];
    CONST robtarget point_711_contact:=[[223,233,134.5],[0,0,1,0],[0, 0, 0, 0],[9E+09,9E+09,9E+09,9E+09,9E+09,9E+09]];
    CONST robtarget point_711_clearance:=[[223,233,149.5],[0,0,1,0],[0, 0, 0, 0],[9E+09,9E+09,9E+09,9E+09,9E+09,9E+09]];
    CONST robtarget point_712_clearance:=[[311,234,149.5],[0,0,1,0],[0, 0, 0, 0],[9E+09,9E+09,9E+09,9E+09,9E+09,9E+09]];
    CONST robtarget point_712_contact:=[[311,234,134.5],[0,0,1,0],[0, 0, 0, 0],[9E+09,9E+09,9E+09,9E+09,9E+09,9E+09]];
    CONST robtarget point_713_contact:=[[288,234,134.5],[0,0,1,0],[0, 0, 0, 0],[9E+09,9E+09,9E+09,9E+09,9E+09,9E+09]];
    CONST robtarget point_713_clearance:=[[288,234,149.5],[0,0,1,0],[0, 0, 0, 0],[9E+09,9E+09,9E+09,9E+09,9E+09,9E+09]];
    CONST robtarget point_714_clearance:=[[345,238,149.5],[0,0,1,0],[0, 0, 0, 0],[9E+09,9E+09,9E+09,9E+09,9E+09,9E+09]];
    CONST robtarget point_714_contact:=[[345,238,134.5],[0,0,1,0],[0, 0, 0, 0],[9E+09,9E+09,9E+09,9E+09,9E+09,9E+09]];
    CONST robtarget point_715_contact:=[[348,234,134.5],[0,0,1,0],[0, 0, 0, 0],[9E+09,9E+09,9E+09,9E+09,9E+09,9E+09]];
    CONST robtarget point_715_clearance:=[[348,234,149.5],[0,0,1,0],[0, 0, 0, 0],[9E+09,9E+09,9E+09,9E+09,9E+09,9E+09]];
    CONST robtarget point_716_clearance:=[[182,235,149.5],[0,0,1,0],[0, 0, 0, 0],[9E+09,9E+09,9E+09,9E+09,9E+09,9E+09]];
    CONST robtarget point_716_contact:=[[182,235,134.5],[0,0,1,0],[0, 0, 0, 0],[9E+09,9E+09,9E+09,9E+09,9E+09,9E+09]];
    CONST robtarget point_717_contact:=[[179,264,134.5],[0,0,1,0],[0, 0, 0, 0],[9E+09,9E+09,9E+09,9E+09,9E+09,9E+09]];
    CONST robtarget point_717_clearance:=[[179,264,149.5],[0,0,1,0],[0, 0, 0, 0],[9E+09,9E+09,9E+09,9E+09,9E+09,9E+09]];
    CONST robtarget point_718_clearance:=[[299,262,149.5],[0,0,1,0],[0, 0, 0, 0],[9E+09,9E+09,9E+09,9E+09,9E+09,9E+09]];
    CONST robtarget point_718_contact:=[[299,262,134.5],[0,0,1,0],[0, 0, 0, 0],[9E+09,9E+09,9E+09,9E+09,9E+09,9E+09]];
    CONST robtarget point_719_contact:=[[270,237,134.5],[0,0,1,0],[0, 0, 0, 0],[9E+09,9E+09,9E+09,9E+09,9E+09,9E+09]];
    CONST robtarget point_719_clearance:=[[270,237,149.5],[0,0,1,0],[0, 0, 0, 0],[9E+09,9E+09,9E+09,9E+09,9E+09,9E+09]];
    CONST robtarget point_720_clearance:=[[433,236,149.5],[0,0,1,0],[0, 0, 0, 0],[9E+09,9E+09,9E+09,9E+09,9E+09,9E+09]];
    CONST robtarget point_720_contact:=[[433,236,134.5],[0,0,1,0],[0, 0, 0, 0],[9E+09,9E+09,9E+09,9E+09,9E+09,9E+09]];
    CONST robtarget point_721_contact:=[[432,252,134.5],[0,0,1,0],[0, 0, 0, 0],[9E+09,9E+09,9E+09,9E+09,9E+09,9E+09]];
    CONST robtarget point_721_clearance:=[[432,252,149.5],[0,0,1,0],[0, 0, 0, 0],[9E+09,9E+09,9E+09,9E+09,9E+09,9E+09]];
    CONST robtarget point_722_clearance:=[[414,237,149.5],[0,0,1,0],[0, 0, 0, 0],[9E+09,9E+09,9E+09,9E+09,9E+09,9E+09]];
    CONST robtarget point_722_contact:=[[414,237,134.5],[0,0,1,0],[0, 0, 0, 0],[9E+09,9E+09,9E+09,9E+09,9E+09,9E+09]];
    CONST robtarget point_723_contact:=[[415,242,134.5],[0,0,1,0],[0, 0, 0, 0],[9E+09,9E+09,9E+09,9E+09,9E+09,9E+09]];
    CONST robtarget point_723_clearance:=[[415,242,149.5],[0,0,1,0],[0, 0, 0, 0],[9E+09,9E+09,9E+09,9E+09,9E+09,9E+09]];
    CONST robtarget point_724_clearance:=[[182,275,149.5],[0,0,1,0],[0, 0, 0, 0],[9E+09,9E+09,9E+09,9E+09,9E+09,9E+09]];
    CONST robtarget point_724_contact:=[[182,275,134.5],[0,0,1,0],[0, 0, 0, 0],[9E+09,9E+09,9E+09,9E+09,9E+09,9E+09]];
    CONST robtarget point_725_contact:=[[185,238,134.5],[0,0,1,0],[0, 0, 0, 0],[9E+09,9E+09,9E+09,9E+09,9E+09,9E+09]];
    CONST robtarget point_725_clearance:=[[185,238,149.5],[0,0,1,0],[0, 0, 0, 0],[9E+09,9E+09,9E+09,9E+09,9E+09,9E+09]];
    CONST robtarget point_726_clearance:=[[400,242,149.5],[0,0,1,0],[0, 0, 0, 0],[9E+09,9E+09,9E+09,9E+09,9E+09,9E+09]];
    CONST robtarget point_726_contact:=[[400,242,134.5],[0,0,1,0],[0, 0, 0, 0],[9E+09,9E+09,9E+09,9E+09,9E+09,9E+09]];
    CONST robtarget point_727_contact:=[[412,242,134.5],[0,0,1,0],[0, 0, 0, 0],[9E+09,9E+09,9E+09,9E+09,9E+09,9E+09]];
    CONST robtarget point_727_clearance:=[[412,242,149.5],[0,0,1,0],[0, 0, 0, 0],[9E+09,9E+09,9E+09,9E+09,9E+09,9E+09]];
    CONST robtarget point_728_clearance:=[[422,239,149.5],[0,0,1,0],[0, 0, 0, 0],[9E+09,9E+09,9E+09,9E+09,9E+09,9E+09]];
    CONST robtarget point_728_contact:=[[422,239,134.5],[0,0,1,0],[0, 0, 0, 0],[9E+09,9E+09,9E+09,9E+09,9E+09,9E+09]];
    CONST robtarget point_729_contact:=[[430,245,134.5],[0,0,1,0],[0, 0, 0, 0],[9E+09,9E+09,9E+09,9E+09,9E+09,9E+09]];
    CONST robtarget point_729_clearance:=[[430,245,149.5],[0,0,1,0],[0, 0, 0, 0],[9E+09,9E+09,9E+09,9E+09,9E+09,9E+09]];
    CONST robtarget point_730_clearance:=[[212,239,149.5],[0,0,1,0],[0, 0, 0, 0],[9E+09,9E+09,9E+09,9E+09,9E+09,9E+09]];
    CONST robtarget point_730_contact:=[[212,239,134.5],[0,0,1,0],[0, 0, 0, 0],[9E+09,9E+09,9E+09,9E+09,9E+09,9E+09]];
    CONST robtarget point_731_contact:=[[218,255,134.5],[0,0,1,0],[0, 0, 0, 0],[9E+09,9E+09,9E+09,9E+09,9E+09,9E+09]];
    CONST robtarget point_731_clearance:=[[218,255,149.5],[0,0,1,0],[0, 0, 0, 0],[9E+09,9E+09,9E+09,9E+09,9E+09,9E+09]];
    CONST robtarget point_732_clearance:=[[338,256,149.5],[0,0,1,0],[0, 0, 0, 0],[9E+09,9E+09,9E+09,9E+09,9E+09,9E+09]];
    CONST robtarget point_732_contact:=[[338,256,134.5],[0,0,1,0],[0, 0, 0, 0],[9E+09,9E+09,9E+09,9E+09,9E+09,9E+09]];
    CONST robtarget point_733_contact:=[[346,239,134.5],[0,0,1,0],[0, 0, 0, 0],[9E+09,9E+09,9E+09,9E+09,9E+09,9E+09]];
    CONST robtarget point_733_clearance:=[[346,239,149.5],[0,0,1,0],[0, 0, 0, 0],[9E+09,9E+09,9E+09,9E+09,9E+09,9E+09]];
    CONST robtarget point_734_clearance:=[[140,243,149.5],[0,0,1,0],[0, 0, 0, 0],[9E+09,9E+09,9E+09,9E+09,9E+09,9E+09]];
    CONST robtarget point_734_contact:=[[140,243,134.5],[0,0,1,0],[0, 0, 0, 0],[9E+09,9E+09,9E+09,9E+09,9E+09,9E+09]];
    CONST robtarget point_735_contact:=[[143,243,134.5],[0,0,1,0],[0, 0, 0, 0],[9E+09,9E+09,9E+09,9E+09,9E+09,9E+09]];
    CONST robtarget point_735_clearance:=[[143,243,149.5],[0,0,1,0],[0, 0, 0, 0],[9E+09,9E+09,9E+09,9E+09,9E+09,9E+09]];
    CONST robtarget point_736_clearance:=[[270,242,149.5],[0,0,1,0],[0, 0, 0, 0],[9E+09,9E+09,9E+09,9E+09,9E+09,9E+09]];
    CONST robtarget point_736_contact:=[[270,242,134.5],[0,0,1,0],[0, 0, 0, 0],[9E+09,9E+09,9E+09,9E+09,9E+09,9E+09]];
    CONST robtarget point_737_contact:=[[271,252,134.5],[0,0,1,0],[0, 0, 0, 0],[9E+09,9E+09,9E+09,9E+09,9E+09,9E+09]];
    CONST robtarget point_737_clearance:=[[271,252,149.5],[0,0,1,0],[0, 0, 0, 0],[9E+09,9E+09,9E+09,9E+09,9E+09,9E+09]];
    CONST robtarget point_738_clearance:=[[390,250,149.5],[0,0,1,0],[0, 0, 0, 0],[9E+09,9E+09,9E+09,9E+09,9E+09,9E+09]];
    CONST robtarget point_738_contact:=[[390,250,134.5],[0,0,1,0],[0, 0, 0, 0],[9E+09,9E+09,9E+09,9E+09,9E+09,9E+09]];
    CONST robtarget point_739_contact:=[[395,242,134.5],[0,0,1,0],[0, 0, 0, 0],[9E+09,9E+09,9E+09,9E+09,9E+09,9E+09]];
    CONST robtarget point_739_clearance:=[[395,242,149.5],[0,0,1,0],[0, 0, 0, 0],[9E+09,9E+09,9E+09,9E+09,9E+09,9E+09]];
    CONST robtarget point_740_clearance:=[[412,246,149.5],[0,0,1,0],[0, 0, 0, 0],[9E+09,9E+09,9E+09,9E+09,9E+09,9E+09]];
    CONST robtarget point_740_contact:=[[412,246,134.5],[0,0,1,0],[0, 0, 0, 0],[9E+09,9E+09,9E+09,9E+09,9E+09,9E+09]];
    CONST robtarget point_741_contact:=[[419,244,134.5],[0,0,1,0],[0, 0, 0, 0],[9E+09,9E+09,9E+09,9E+09,9E+09,9E+09]];
    CONST robtarget point_741_clearance:=[[419,244,149.5],[0,0,1,0],[0, 0, 0, 0],[9E+09,9E+09,9E+09,9E+09,9E+09,9E+09]];
    CONST robtarget point_742_clearance:=[[419,247,149.5],[0,0,1,0],[0, 0, 0, 0],[9E+09,9E+09,9E+09,9E+09,9E+09,9E+09]];
    CONST robtarget point_742_contact:=[[419,247,134.5],[0,0,1,0],[0, 0, 0, 0],[9E+09,9E+09,9E+09,9E+09,9E+09,9E+09]];
    CONST robtarget point_743_contact:=[[424,243,134.5],[0,0,1,0],[0, 0, 0, 0],[9E+09,9E+09,9E+09,9E+09,9E+09,9E+09]];
    CONST robtarget point_743_clearance:=[[424,243,149.5],[0,0,1,0],[0, 0, 0, 0],[9E+09,9E+09,9E+09,9E+09,9E+09,9E+09]];
    CONST robtarget point_744_clearance:=[[142,245,149.5],[0,0,1,0],[0, 0, 0, 0],[9E+09,9E+09,9E+09,9E+09,9E+09,9E+09]];
    CONST robtarget point_744_contact:=[[142,245,134.5],[0,0,1,0],[0, 0, 0, 0],[9E+09,9E+09,9E+09,9E+09,9E+09,9E+09]];
    CONST robtarget point_745_contact:=[[152,245,134.5],[0,0,1,0],[0, 0, 0, 0],[9E+09,9E+09,9E+09,9E+09,9E+09,9E+09]];
    CONST robtarget point_745_clearance:=[[152,245,149.5],[0,0,1,0],[0, 0, 0, 0],[9E+09,9E+09,9E+09,9E+09,9E+09,9E+09]];
    CONST robtarget point_746_clearance:=[[225,251,149.5],[0,0,1,0],[0, 0, 0, 0],[9E+09,9E+09,9E+09,9E+09,9E+09,9E+09]];
    CONST robtarget point_746_contact:=[[225,251,134.5],[0,0,1,0],[0, 0, 0, 0],[9E+09,9E+09,9E+09,9E+09,9E+09,9E+09]];
    CONST robtarget point_747_contact:=[[221,243,134.5],[0,0,1,0],[0, 0, 0, 0],[9E+09,9E+09,9E+09,9E+09,9E+09,9E+09]];
    CONST robtarget point_747_clearance:=[[221,243,149.5],[0,0,1,0],[0, 0, 0, 0],[9E+09,9E+09,9E+09,9E+09,9E+09,9E+09]];
    CONST robtarget point_748_clearance:=[[234,244,149.5],[0,0,1,0],[0, 0, 0, 0],[9E+09,9E+09,9E+09,9E+09,9E+09,9E+09]];
    CONST robtarget point_748_contact:=[[234,244,134.5],[0,0,1,0],[0, 0, 0, 0],[9E+09,9E+09,9E+09,9E+09,9E+09,9E+09]];
    CONST robtarget point_749_contact:=[[228,254,134.5],[0,0,1,0],[0, 0, 0, 0],[9E+09,9E+09,9E+09,9E+09,9E+09,9E+09]];
    CONST robtarget point_749_clearance:=[[228,254,149.5],[0,0,1,0],[0, 0, 0, 0],[9E+09,9E+09,9E+09,9E+09,9E+09,9E+09]];
    CONST robtarget point_750_clearance:=[[295,247,149.5],[0,0,1,0],[0, 0, 0, 0],[9E+09,9E+09,9E+09,9E+09,9E+09,9E+09]];
    CONST robtarget point_750_contact:=[[295,247,134.5],[0,0,1,0],[0, 0, 0, 0],[9E+09,9E+09,9E+09,9E+09,9E+09,9E+09]];
    CONST robtarget point_751_contact:=[[283,244,134.5],[0,0,1,0],[0, 0, 0, 0],[9E+09,9E+09,9E+09,9E+09,9E+09,9E+09]];
    CONST robtarget point_751_clearance:=[[283,244,149.5],[0,0,1,0],[0, 0, 0, 0],[9E+09,9E+09,9E+09,9E+09,9E+09,9E+09]];
    CONST robtarget point_752_clearance:=[[237,245,149.5],[0,0,1,0],[0, 0, 0, 0],[9E+09,9E+09,9E+09,9E+09,9E+09,9E+09]];
    CONST robtarget point_752_contact:=[[237,245,134.5],[0,0,1,0],[0, 0, 0, 0],[9E+09,9E+09,9E+09,9E+09,9E+09,9E+09]];
    CONST robtarget point_753_contact:=[[245,258,134.5],[0,0,1,0],[0, 0, 0, 0],[9E+09,9E+09,9E+09,9E+09,9E+09,9E+09]];
    CONST robtarget point_753_clearance:=[[245,258,149.5],[0,0,1,0],[0, 0, 0, 0],[9E+09,9E+09,9E+09,9E+09,9E+09,9E+09]];
    CONST robtarget point_754_clearance:=[[155,250,149.5],[0,0,1,0],[0, 0, 0, 0],[9E+09,9E+09,9E+09,9E+09,9E+09,9E+09]];
    CONST robtarget point_754_contact:=[[155,250,134.5],[0,0,1,0],[0, 0, 0, 0],[9E+09,9E+09,9E+09,9E+09,9E+09,9E+09]];
    CONST robtarget point_755_contact:=[[175,246,134.5],[0,0,1,0],[0, 0, 0, 0],[9E+09,9E+09,9E+09,9E+09,9E+09,9E+09]];
    CONST robtarget point_755_clearance:=[[175,246,149.5],[0,0,1,0],[0, 0, 0, 0],[9E+09,9E+09,9E+09,9E+09,9E+09,9E+09]];
    CONST robtarget point_756_clearance:=[[195,246,149.5],[0,0,1,0],[0, 0, 0, 0],[9E+09,9E+09,9E+09,9E+09,9E+09,9E+09]];
    CONST robtarget point_756_contact:=[[195,246,134.5],[0,0,1,0],[0, 0, 0, 0],[9E+09,9E+09,9E+09,9E+09,9E+09,9E+09]];
    CONST robtarget point_757_contact:=[[197,267,134.5],[0,0,1,0],[0, 0, 0, 0],[9E+09,9E+09,9E+09,9E+09,9E+09,9E+09]];
    CONST robtarget point_757_clearance:=[[197,267,149.5],[0,0,1,0],[0, 0, 0, 0],[9E+09,9E+09,9E+09,9E+09,9E+09,9E+09]];
    CONST robtarget point_758_clearance:=[[417,248,149.5],[0,0,1,0],[0, 0, 0, 0],[9E+09,9E+09,9E+09,9E+09,9E+09,9E+09]];
    CONST robtarget point_758_contact:=[[417,248,134.5],[0,0,1,0],[0, 0, 0, 0],[9E+09,9E+09,9E+09,9E+09,9E+09,9E+09]];
    CONST robtarget point_759_contact:=[[425,252,134.5],[0,0,1,0],[0, 0, 0, 0],[9E+09,9E+09,9E+09,9E+09,9E+09,9E+09]];
    CONST robtarget point_759_clearance:=[[425,252,149.5],[0,0,1,0],[0, 0, 0, 0],[9E+09,9E+09,9E+09,9E+09,9E+09,9E+09]];
    CONST robtarget point_760_clearance:=[[190,268,149.5],[0,0,1,0],[0, 0, 0, 0],[9E+09,9E+09,9E+09,9E+09,9E+09,9E+09]];
    CONST robtarget point_760_contact:=[[190,268,134.5],[0,0,1,0],[0, 0, 0, 0],[9E+09,9E+09,9E+09,9E+09,9E+09,9E+09]];
    CONST robtarget point_761_contact:=[[192,247,134.5],[0,0,1,0],[0, 0, 0, 0],[9E+09,9E+09,9E+09,9E+09,9E+09,9E+09]];
    CONST robtarget point_761_clearance:=[[192,247,149.5],[0,0,1,0],[0, 0, 0, 0],[9E+09,9E+09,9E+09,9E+09,9E+09,9E+09]];
    CONST robtarget point_762_clearance:=[[380,256,149.5],[0,0,1,0],[0, 0, 0, 0],[9E+09,9E+09,9E+09,9E+09,9E+09,9E+09]];
    CONST robtarget point_762_contact:=[[380,256,134.5],[0,0,1,0],[0, 0, 0, 0],[9E+09,9E+09,9E+09,9E+09,9E+09,9E+09]];
    CONST robtarget point_763_contact:=[[389,250,134.5],[0,0,1,0],[0, 0, 0, 0],[9E+09,9E+09,9E+09,9E+09,9E+09,9E+09]];
    CONST robtarget point_763_clearance:=[[389,250,149.5],[0,0,1,0],[0, 0, 0, 0],[9E+09,9E+09,9E+09,9E+09,9E+09,9E+09]];
    CONST robtarget point_764_clearance:=[[225,257,149.5],[0,0,1,0],[0, 0, 0, 0],[9E+09,9E+09,9E+09,9E+09,9E+09,9E+09]];
    CONST robtarget point_764_contact:=[[225,257,134.5],[0,0,1,0],[0, 0, 0, 0],[9E+09,9E+09,9E+09,9E+09,9E+09,9E+09]];
    CONST robtarget point_765_contact:=[[225,252,134.5],[0,0,1,0],[0, 0, 0, 0],[9E+09,9E+09,9E+09,9E+09,9E+09,9E+09]];
    CONST robtarget point_765_clearance:=[[225,252,149.5],[0,0,1,0],[0, 0, 0, 0],[9E+09,9E+09,9E+09,9E+09,9E+09,9E+09]];
    CONST robtarget point_766_clearance:=[[265,275,149.5],[0,0,1,0],[0, 0, 0, 0],[9E+09,9E+09,9E+09,9E+09,9E+09,9E+09]];
    CONST robtarget point_766_contact:=[[265,275,134.5],[0,0,1,0],[0, 0, 0, 0],[9E+09,9E+09,9E+09,9E+09,9E+09,9E+09]];
    CONST robtarget point_767_contact:=[[261,252,134.5],[0,0,1,0],[0, 0, 0, 0],[9E+09,9E+09,9E+09,9E+09,9E+09,9E+09]];
    CONST robtarget point_767_clearance:=[[261,252,149.5],[0,0,1,0],[0, 0, 0, 0],[9E+09,9E+09,9E+09,9E+09,9E+09,9E+09]];
    CONST robtarget point_768_clearance:=[[271,252,149.5],[0,0,1,0],[0, 0, 0, 0],[9E+09,9E+09,9E+09,9E+09,9E+09,9E+09]];
    CONST robtarget point_768_contact:=[[271,252,134.5],[0,0,1,0],[0, 0, 0, 0],[9E+09,9E+09,9E+09,9E+09,9E+09,9E+09]];
    CONST robtarget point_769_contact:=[[277,274,134.5],[0,0,1,0],[0, 0, 0, 0],[9E+09,9E+09,9E+09,9E+09,9E+09,9E+09]];
    CONST robtarget point_769_clearance:=[[277,274,149.5],[0,0,1,0],[0, 0, 0, 0],[9E+09,9E+09,9E+09,9E+09,9E+09,9E+09]];
    CONST robtarget point_770_clearance:=[[421,252,149.5],[0,0,1,0],[0, 0, 0, 0],[9E+09,9E+09,9E+09,9E+09,9E+09,9E+09]];
    CONST robtarget point_770_contact:=[[421,252,134.5],[0,0,1,0],[0, 0, 0, 0],[9E+09,9E+09,9E+09,9E+09,9E+09,9E+09]];
    CONST robtarget point_771_contact:=[[435,255,134.5],[0,0,1,0],[0, 0, 0, 0],[9E+09,9E+09,9E+09,9E+09,9E+09,9E+09]];
    CONST robtarget point_771_clearance:=[[435,255,149.5],[0,0,1,0],[0, 0, 0, 0],[9E+09,9E+09,9E+09,9E+09,9E+09,9E+09]];
    CONST robtarget point_772_clearance:=[[256,253,149.5],[0,0,1,0],[0, 0, 0, 0],[9E+09,9E+09,9E+09,9E+09,9E+09,9E+09]];
    CONST robtarget point_772_contact:=[[256,253,134.5],[0,0,1,0],[0, 0, 0, 0],[9E+09,9E+09,9E+09,9E+09,9E+09,9E+09]];
    CONST robtarget point_773_contact:=[[256,270,134.5],[0,0,1,0],[0, 0, 0, 0],[9E+09,9E+09,9E+09,9E+09,9E+09,9E+09]];
    CONST robtarget point_773_clearance:=[[256,270,149.5],[0,0,1,0],[0, 0, 0, 0],[9E+09,9E+09,9E+09,9E+09,9E+09,9E+09]];
    CONST robtarget point_774_clearance:=[[225,258,149.5],[0,0,1,0],[0, 0, 0, 0],[9E+09,9E+09,9E+09,9E+09,9E+09,9E+09]];
    CONST robtarget point_774_contact:=[[225,258,134.5],[0,0,1,0],[0, 0, 0, 0],[9E+09,9E+09,9E+09,9E+09,9E+09,9E+09]];
    CONST robtarget point_775_contact:=[[235,257,134.5],[0,0,1,0],[0, 0, 0, 0],[9E+09,9E+09,9E+09,9E+09,9E+09,9E+09]];
    CONST robtarget point_775_clearance:=[[235,257,149.5],[0,0,1,0],[0, 0, 0, 0],[9E+09,9E+09,9E+09,9E+09,9E+09,9E+09]];
    CONST robtarget point_776_clearance:=[[218,256,149.5],[0,0,1,0],[0, 0, 0, 0],[9E+09,9E+09,9E+09,9E+09,9E+09,9E+09]];
    CONST robtarget point_776_contact:=[[218,256,134.5],[0,0,1,0],[0, 0, 0, 0],[9E+09,9E+09,9E+09,9E+09,9E+09,9E+09]];
    CONST robtarget point_777_contact:=[[215,260,134.5],[0,0,1,0],[0, 0, 0, 0],[9E+09,9E+09,9E+09,9E+09,9E+09,9E+09]];
    CONST robtarget point_777_clearance:=[[215,260,149.5],[0,0,1,0],[0, 0, 0, 0],[9E+09,9E+09,9E+09,9E+09,9E+09,9E+09]];
    CONST robtarget point_778_clearance:=[[218,256,149.5],[0,0,1,0],[0, 0, 0, 0],[9E+09,9E+09,9E+09,9E+09,9E+09,9E+09]];
    CONST robtarget point_778_contact:=[[218,256,134.5],[0,0,1,0],[0, 0, 0, 0],[9E+09,9E+09,9E+09,9E+09,9E+09,9E+09]];
    CONST robtarget point_779_contact:=[[223,275,134.5],[0,0,1,0],[0, 0, 0, 0],[9E+09,9E+09,9E+09,9E+09,9E+09,9E+09]];
    CONST robtarget point_779_clearance:=[[223,275,149.5],[0,0,1,0],[0, 0, 0, 0],[9E+09,9E+09,9E+09,9E+09,9E+09,9E+09]];
    CONST robtarget point_780_clearance:=[[246,258,149.5],[0,0,1,0],[0, 0, 0, 0],[9E+09,9E+09,9E+09,9E+09,9E+09,9E+09]];
    CONST robtarget point_780_contact:=[[246,258,134.5],[0,0,1,0],[0, 0, 0, 0],[9E+09,9E+09,9E+09,9E+09,9E+09,9E+09]];
    CONST robtarget point_781_contact:=[[268,290,134.5],[0,0,1,0],[0, 0, 0, 0],[9E+09,9E+09,9E+09,9E+09,9E+09,9E+09]];
    CONST robtarget point_781_clearance:=[[268,290,149.5],[0,0,1,0],[0, 0, 0, 0],[9E+09,9E+09,9E+09,9E+09,9E+09,9E+09]];
    CONST robtarget point_782_clearance:=[[227,263,149.5],[0,0,1,0],[0, 0, 0, 0],[9E+09,9E+09,9E+09,9E+09,9E+09,9E+09]];
    CONST robtarget point_782_contact:=[[227,263,134.5],[0,0,1,0],[0, 0, 0, 0],[9E+09,9E+09,9E+09,9E+09,9E+09,9E+09]];
    CONST robtarget point_783_contact:=[[238,262,134.5],[0,0,1,0],[0, 0, 0, 0],[9E+09,9E+09,9E+09,9E+09,9E+09,9E+09]];
    CONST robtarget point_783_clearance:=[[238,262,149.5],[0,0,1,0],[0, 0, 0, 0],[9E+09,9E+09,9E+09,9E+09,9E+09,9E+09]];
    CONST robtarget point_784_clearance:=[[329,274,149.5],[0,0,1,0],[0, 0, 0, 0],[9E+09,9E+09,9E+09,9E+09,9E+09,9E+09]];
    CONST robtarget point_784_contact:=[[329,274,134.5],[0,0,1,0],[0, 0, 0, 0],[9E+09,9E+09,9E+09,9E+09,9E+09,9E+09]];
    CONST robtarget point_785_contact:=[[299,263,134.5],[0,0,1,0],[0, 0, 0, 0],[9E+09,9E+09,9E+09,9E+09,9E+09,9E+09]];
    CONST robtarget point_785_clearance:=[[299,263,149.5],[0,0,1,0],[0, 0, 0, 0],[9E+09,9E+09,9E+09,9E+09,9E+09,9E+09]];
    CONST robtarget point_786_clearance:=[[209,268,149.5],[0,0,1,0],[0, 0, 0, 0],[9E+09,9E+09,9E+09,9E+09,9E+09,9E+09]];
    CONST robtarget point_786_contact:=[[209,268,134.5],[0,0,1,0],[0, 0, 0, 0],[9E+09,9E+09,9E+09,9E+09,9E+09,9E+09]];
    CONST robtarget point_787_contact:=[[218,264,134.5],[0,0,1,0],[0, 0, 0, 0],[9E+09,9E+09,9E+09,9E+09,9E+09,9E+09]];
    CONST robtarget point_787_clearance:=[[218,264,149.5],[0,0,1,0],[0, 0, 0, 0],[9E+09,9E+09,9E+09,9E+09,9E+09,9E+09]];
    CONST robtarget point_788_clearance:=[[179,265,149.5],[0,0,1,0],[0, 0, 0, 0],[9E+09,9E+09,9E+09,9E+09,9E+09,9E+09]];
    CONST robtarget point_788_contact:=[[179,265,134.5],[0,0,1,0],[0, 0, 0, 0],[9E+09,9E+09,9E+09,9E+09,9E+09,9E+09]];
    CONST robtarget point_789_contact:=[[178,273,134.5],[0,0,1,0],[0, 0, 0, 0],[9E+09,9E+09,9E+09,9E+09,9E+09,9E+09]];
    CONST robtarget point_789_clearance:=[[178,273,149.5],[0,0,1,0],[0, 0, 0, 0],[9E+09,9E+09,9E+09,9E+09,9E+09,9E+09]];
    CONST robtarget point_790_clearance:=[[200,267,149.5],[0,0,1,0],[0, 0, 0, 0],[9E+09,9E+09,9E+09,9E+09,9E+09,9E+09]];
    CONST robtarget point_790_contact:=[[200,267,134.5],[0,0,1,0],[0, 0, 0, 0],[9E+09,9E+09,9E+09,9E+09,9E+09,9E+09]];
    CONST robtarget point_791_contact:=[[207,269,134.5],[0,0,1,0],[0, 0, 0, 0],[9E+09,9E+09,9E+09,9E+09,9E+09,9E+09]];
    CONST robtarget point_791_clearance:=[[207,269,149.5],[0,0,1,0],[0, 0, 0, 0],[9E+09,9E+09,9E+09,9E+09,9E+09,9E+09]];
    CONST robtarget point_792_clearance:=[[228,265,149.5],[0,0,1,0],[0, 0, 0, 0],[9E+09,9E+09,9E+09,9E+09,9E+09,9E+09]];
    CONST robtarget point_792_contact:=[[228,265,134.5],[0,0,1,0],[0, 0, 0, 0],[9E+09,9E+09,9E+09,9E+09,9E+09,9E+09]];
    CONST robtarget point_793_contact:=[[231,268,134.5],[0,0,1,0],[0, 0, 0, 0],[9E+09,9E+09,9E+09,9E+09,9E+09,9E+09]];
    CONST robtarget point_793_clearance:=[[231,268,149.5],[0,0,1,0],[0, 0, 0, 0],[9E+09,9E+09,9E+09,9E+09,9E+09,9E+09]];
    CONST robtarget point_794_clearance:=[[232,270,149.5],[0,0,1,0],[0, 0, 0, 0],[9E+09,9E+09,9E+09,9E+09,9E+09,9E+09]];
    CONST robtarget point_794_contact:=[[232,270,134.5],[0,0,1,0],[0, 0, 0, 0],[9E+09,9E+09,9E+09,9E+09,9E+09,9E+09]];
    CONST robtarget point_795_contact:=[[238,265,134.5],[0,0,1,0],[0, 0, 0, 0],[9E+09,9E+09,9E+09,9E+09,9E+09,9E+09]];
    CONST robtarget point_795_clearance:=[[238,265,149.5],[0,0,1,0],[0, 0, 0, 0],[9E+09,9E+09,9E+09,9E+09,9E+09,9E+09]];
    CONST robtarget point_796_clearance:=[[228,271,149.5],[0,0,1,0],[0, 0, 0, 0],[9E+09,9E+09,9E+09,9E+09,9E+09,9E+09]];
    CONST robtarget point_796_contact:=[[228,271,134.5],[0,0,1,0],[0, 0, 0, 0],[9E+09,9E+09,9E+09,9E+09,9E+09,9E+09]];
    CONST robtarget point_797_contact:=[[236,271,134.5],[0,0,1,0],[0, 0, 0, 0],[9E+09,9E+09,9E+09,9E+09,9E+09,9E+09]];
    CONST robtarget point_797_clearance:=[[236,271,149.5],[0,0,1,0],[0, 0, 0, 0],[9E+09,9E+09,9E+09,9E+09,9E+09,9E+09]];
    CONST robtarget point_798_clearance:=[[327,274,149.5],[0,0,1,0],[0, 0, 0, 0],[9E+09,9E+09,9E+09,9E+09,9E+09,9E+09]];
    CONST robtarget point_798_contact:=[[327,274,134.5],[0,0,1,0],[0, 0, 0, 0],[9E+09,9E+09,9E+09,9E+09,9E+09,9E+09]];
    CONST robtarget point_799_contact:=[[338,272,134.5],[0,0,1,0],[0, 0, 0, 0],[9E+09,9E+09,9E+09,9E+09,9E+09,9E+09]];
    CONST robtarget point_799_clearance:=[[338,272,149.5],[0,0,1,0],[0, 0, 0, 0],[9E+09,9E+09,9E+09,9E+09,9E+09,9E+09]];
    CONST robtarget point_800_clearance:=[[277,275,149.5],[0,0,1,0],[0, 0, 0, 0],[9E+09,9E+09,9E+09,9E+09,9E+09,9E+09]];
    CONST robtarget point_800_contact:=[[277,275,134.5],[0,0,1,0],[0, 0, 0, 0],[9E+09,9E+09,9E+09,9E+09,9E+09,9E+09]];
    CONST robtarget point_801_contact:=[[278,285,134.5],[0,0,1,0],[0, 0, 0, 0],[9E+09,9E+09,9E+09,9E+09,9E+09,9E+09]];
    CONST robtarget point_801_clearance:=[[278,285,149.5],[0,0,1,0],[0, 0, 0, 0],[9E+09,9E+09,9E+09,9E+09,9E+09,9E+09]];
    CONST robtarget point_802_clearance:=[[336,275,149.5],[0,0,1,0],[0, 0, 0, 0],[9E+09,9E+09,9E+09,9E+09,9E+09,9E+09]];
    CONST robtarget point_802_contact:=[[336,275,134.5],[0,0,1,0],[0, 0, 0, 0],[9E+09,9E+09,9E+09,9E+09,9E+09,9E+09]];
    CONST robtarget point_803_contact:=[[308,298,134.5],[0,0,1,0],[0, 0, 0, 0],[9E+09,9E+09,9E+09,9E+09,9E+09,9E+09]];
    CONST robtarget point_803_clearance:=[[308,298,149.5],[0,0,1,0],[0, 0, 0, 0],[9E+09,9E+09,9E+09,9E+09,9E+09,9E+09]];
    CONST robtarget point_804_clearance:=[[269,278,149.5],[0,0,1,0],[0, 0, 0, 0],[9E+09,9E+09,9E+09,9E+09,9E+09,9E+09]];
    CONST robtarget point_804_contact:=[[269,278,134.5],[0,0,1,0],[0, 0, 0, 0],[9E+09,9E+09,9E+09,9E+09,9E+09,9E+09]];
    CONST robtarget point_805_contact:=[[277,287,134.5],[0,0,1,0],[0, 0, 0, 0],[9E+09,9E+09,9E+09,9E+09,9E+09,9E+09]];
    CONST robtarget point_805_clearance:=[[277,287,149.5],[0,0,1,0],[0, 0, 0, 0],[9E+09,9E+09,9E+09,9E+09,9E+09,9E+09]];
    CONST robtarget point_806_clearance:=[[297,303,149.5],[0,0,1,0],[0, 0, 0, 0],[9E+09,9E+09,9E+09,9E+09,9E+09,9E+09]];
    CONST robtarget point_806_contact:=[[297,303,134.5],[0,0,1,0],[0, 0, 0, 0],[9E+09,9E+09,9E+09,9E+09,9E+09,9E+09]];
    CONST robtarget point_807_contact:=[[331,277,134.5],[0,0,1,0],[0, 0, 0, 0],[9E+09,9E+09,9E+09,9E+09,9E+09,9E+09]];
    CONST robtarget point_807_clearance:=[[331,277,149.5],[0,0,1,0],[0, 0, 0, 0],[9E+09,9E+09,9E+09,9E+09,9E+09,9E+09]];
    CONST robtarget point_808_clearance:=[[176,279,149.5],[0,0,1,0],[0, 0, 0, 0],[9E+09,9E+09,9E+09,9E+09,9E+09,9E+09]];
    CONST robtarget point_808_contact:=[[176,279,134.5],[0,0,1,0],[0, 0, 0, 0],[9E+09,9E+09,9E+09,9E+09,9E+09,9E+09]];
    CONST robtarget point_809_contact:=[[166,286,134.5],[0,0,1,0],[0, 0, 0, 0],[9E+09,9E+09,9E+09,9E+09,9E+09,9E+09]];
    CONST robtarget point_809_clearance:=[[166,286,149.5],[0,0,1,0],[0, 0, 0, 0],[9E+09,9E+09,9E+09,9E+09,9E+09,9E+09]];
    CONST robtarget point_810_clearance:=[[292,318,149.5],[0,0,1,0],[0, 0, 0, 0],[9E+09,9E+09,9E+09,9E+09,9E+09,9E+09]];
    CONST robtarget point_810_contact:=[[292,318,134.5],[0,0,1,0],[0, 0, 0, 0],[9E+09,9E+09,9E+09,9E+09,9E+09,9E+09]];
    CONST robtarget point_811_contact:=[[337,278,134.5],[0,0,1,0],[0, 0, 0, 0],[9E+09,9E+09,9E+09,9E+09,9E+09,9E+09]];
    CONST robtarget point_811_clearance:=[[337,278,149.5],[0,0,1,0],[0, 0, 0, 0],[9E+09,9E+09,9E+09,9E+09,9E+09,9E+09]];
    CONST robtarget point_812_clearance:=[[168,289,149.5],[0,0,1,0],[0, 0, 0, 0],[9E+09,9E+09,9E+09,9E+09,9E+09,9E+09]];
    CONST robtarget point_812_contact:=[[168,289,134.5],[0,0,1,0],[0, 0, 0, 0],[9E+09,9E+09,9E+09,9E+09,9E+09,9E+09]];
    CONST robtarget point_813_contact:=[[178,281,134.5],[0,0,1,0],[0, 0, 0, 0],[9E+09,9E+09,9E+09,9E+09,9E+09,9E+09]];
    CONST robtarget point_813_clearance:=[[178,281,149.5],[0,0,1,0],[0, 0, 0, 0],[9E+09,9E+09,9E+09,9E+09,9E+09,9E+09]];
    CONST robtarget point_814_clearance:=[[280,284,149.5],[0,0,1,0],[0, 0, 0, 0],[9E+09,9E+09,9E+09,9E+09,9E+09,9E+09]];
    CONST robtarget point_814_contact:=[[280,284,134.5],[0,0,1,0],[0, 0, 0, 0],[9E+09,9E+09,9E+09,9E+09,9E+09,9E+09]];
    CONST robtarget point_815_contact:=[[279,292,134.5],[0,0,1,0],[0, 0, 0, 0],[9E+09,9E+09,9E+09,9E+09,9E+09,9E+09]];
    CONST robtarget point_815_clearance:=[[279,292,149.5],[0,0,1,0],[0, 0, 0, 0],[9E+09,9E+09,9E+09,9E+09,9E+09,9E+09]];
    CONST robtarget point_816_clearance:=[[280,290,149.5],[0,0,1,0],[0, 0, 0, 0],[9E+09,9E+09,9E+09,9E+09,9E+09,9E+09]];
    CONST robtarget point_816_contact:=[[280,290,134.5],[0,0,1,0],[0, 0, 0, 0],[9E+09,9E+09,9E+09,9E+09,9E+09,9E+09]];
    CONST robtarget point_817_contact:=[[292,301,134.5],[0,0,1,0],[0, 0, 0, 0],[9E+09,9E+09,9E+09,9E+09,9E+09,9E+09]];
    CONST robtarget point_817_clearance:=[[292,301,149.5],[0,0,1,0],[0, 0, 0, 0],[9E+09,9E+09,9E+09,9E+09,9E+09,9E+09]];
    CONST robtarget point_818_clearance:=[[268,291,149.5],[0,0,1,0],[0, 0, 0, 0],[9E+09,9E+09,9E+09,9E+09,9E+09,9E+09]];
    CONST robtarget point_818_contact:=[[268,291,134.5],[0,0,1,0],[0, 0, 0, 0],[9E+09,9E+09,9E+09,9E+09,9E+09,9E+09]];
    CONST robtarget point_819_contact:=[[276,301,134.5],[0,0,1,0],[0, 0, 0, 0],[9E+09,9E+09,9E+09,9E+09,9E+09,9E+09]];
    CONST robtarget point_819_clearance:=[[276,301,149.5],[0,0,1,0],[0, 0, 0, 0],[9E+09,9E+09,9E+09,9E+09,9E+09,9E+09]];
    CONST robtarget point_820_clearance:=[[293,305,149.5],[0,0,1,0],[0, 0, 0, 0],[9E+09,9E+09,9E+09,9E+09,9E+09,9E+09]];
    CONST robtarget point_820_contact:=[[293,305,134.5],[0,0,1,0],[0, 0, 0, 0],[9E+09,9E+09,9E+09,9E+09,9E+09,9E+09]];
    CONST robtarget point_821_contact:=[[283,297,134.5],[0,0,1,0],[0, 0, 0, 0],[9E+09,9E+09,9E+09,9E+09,9E+09,9E+09]];
    CONST robtarget point_821_clearance:=[[283,297,149.5],[0,0,1,0],[0, 0, 0, 0],[9E+09,9E+09,9E+09,9E+09,9E+09,9E+09]];
    CONST robtarget point_822_clearance:=[[277,299,149.5],[0,0,1,0],[0, 0, 0, 0],[9E+09,9E+09,9E+09,9E+09,9E+09,9E+09]];
    CONST robtarget point_822_contact:=[[277,299,134.5],[0,0,1,0],[0, 0, 0, 0],[9E+09,9E+09,9E+09,9E+09,9E+09,9E+09]];
    CONST robtarget point_823_contact:=[[289,319,134.5],[0,0,1,0],[0, 0, 0, 0],[9E+09,9E+09,9E+09,9E+09,9E+09,9E+09]];
    CONST robtarget point_823_clearance:=[[289,319,149.5],[0,0,1,0],[0, 0, 0, 0],[9E+09,9E+09,9E+09,9E+09,9E+09,9E+09]];
    CONST robtarget point_824_clearance:=[[291,312,149.5],[0,0,1,0],[0, 0, 0, 0],[9E+09,9E+09,9E+09,9E+09,9E+09,9E+09]];
    CONST robtarget point_824_contact:=[[291,312,134.5],[0,0,1,0],[0, 0, 0, 0],[9E+09,9E+09,9E+09,9E+09,9E+09,9E+09]];
    CONST robtarget point_825_contact:=[[294,304,134.5],[0,0,1,0],[0, 0, 0, 0],[9E+09,9E+09,9E+09,9E+09,9E+09,9E+09]];
    CONST robtarget point_825_clearance:=[[294,304,149.5],[0,0,1,0],[0, 0, 0, 0],[9E+09,9E+09,9E+09,9E+09,9E+09,9E+09]];



    PROC main()
        Path_Calib;
        Path_Draw;
    ENDPROC
    LOCAL PROC Path_Calib()
        MoveAbsJ home,v500,fine,GS25_ParallelGripper\WObj:=Workobject_1;
        MoveL calib_1,v500,fine,GS25_ParallelGripper\WObj:=Workobject_1;
        MoveL calib_1d,v100,fine,GS25_ParallelGripper\WObj:=Workobject_1;
        MoveL calib_1,v100,fine,GS25_ParallelGripper\WObj:=Workobject_1;
        MoveL calib_2,v100,fine,GS25_ParallelGripper\WObj:=Workobject_1;
        MoveL calib_2d,v100,fine,GS25_ParallelGripper\WObj:=Workobject_1;
        MoveL calib_2,v100,fine,GS25_ParallelGripper\WObj:=Workobject_1;
        MoveL calib_3,v100,fine,GS25_ParallelGripper\WObj:=Workobject_1;
        MoveL calib_3d,v100,fine,GS25_ParallelGripper\WObj:=Workobject_1;
        MoveL calib_3,v100,fine,GS25_ParallelGripper\WObj:=Workobject_1;
        MoveL calib_4,v100,fine,GS25_ParallelGripper\WObj:=Workobject_1;
        MoveL calib_4d,v100,fine,GS25_ParallelGripper\WObj:=Workobject_1;
        MoveL calib_4,v100,fine,GS25_ParallelGripper\WObj:=Workobject_1;
        MoveL calib_1,v100,fine,GS25_ParallelGripper\WObj:=Workobject_1;
    ENDPROC

